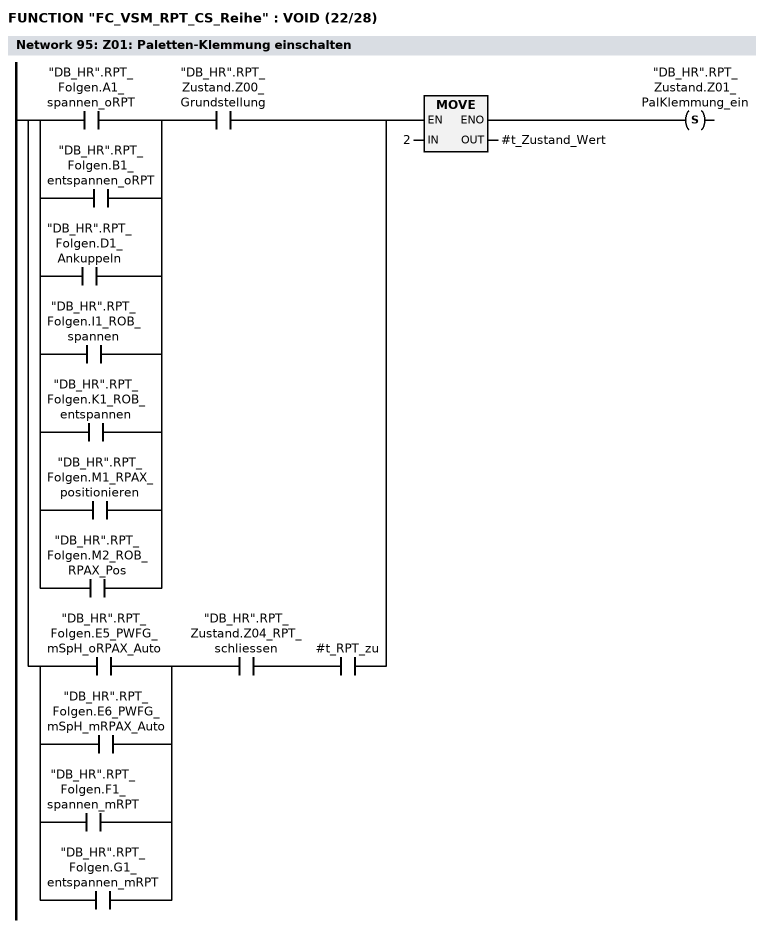

      U(    ;
      U(    ;
      O     "DB_HR".RPT_Folgen.A1_spannen_oRPT;
      O     "DB_HR".RPT_Folgen.B1_entspannen_oRPT;
      O     "DB_HR".RPT_Folgen.D1_Ankuppeln;
      O     "DB_HR".RPT_Folgen.I1_ROB_spannen;
      O     "DB_HR".RPT_Folgen.K1_ROB_entspannen;
      O     "DB_HR".RPT_Folgen.M1_RPAX_positionieren;
//      O     "DB_HR".RPT_Folgen.L2_ROB_PWFG_mRPAX
      O     "DB_HR".RPT_Folgen.M2_ROB_RPAX_Pos;
      )     ;
      U     "DB_HR".RPT_Zustand.Z00_Grundstellung;
      O     ;
      U(    ;
      O     "DB_HR".RPT_Folgen.E5_PWFG_mSpH_oRPAX_Auto;
      O     "DB_HR".RPT_Folgen.E6_PWFG_mSpH_mRPAX_Auto;
      O     "DB_HR".RPT_Folgen.F1_spannen_mRPT;
      O     "DB_HR".RPT_Folgen.G1_entspannen_mRPT;
      )     ;
      U     "DB_HR".RPT_Zustand.Z04_RPT_schliessen;
      U     #t_RPT_zu;
      )     ;
      SPBNB _01d;
      L     2;
      T     #t_Zustand_Wert;
      SET   ;
      SAVE  ;
      CLR   ;
_01d: U     BIE;
      S     "DB_HR".RPT_Zustand.Z01_PalKlemmung_ein;
NETWORK
TITLE =Z02: Ankuppeln
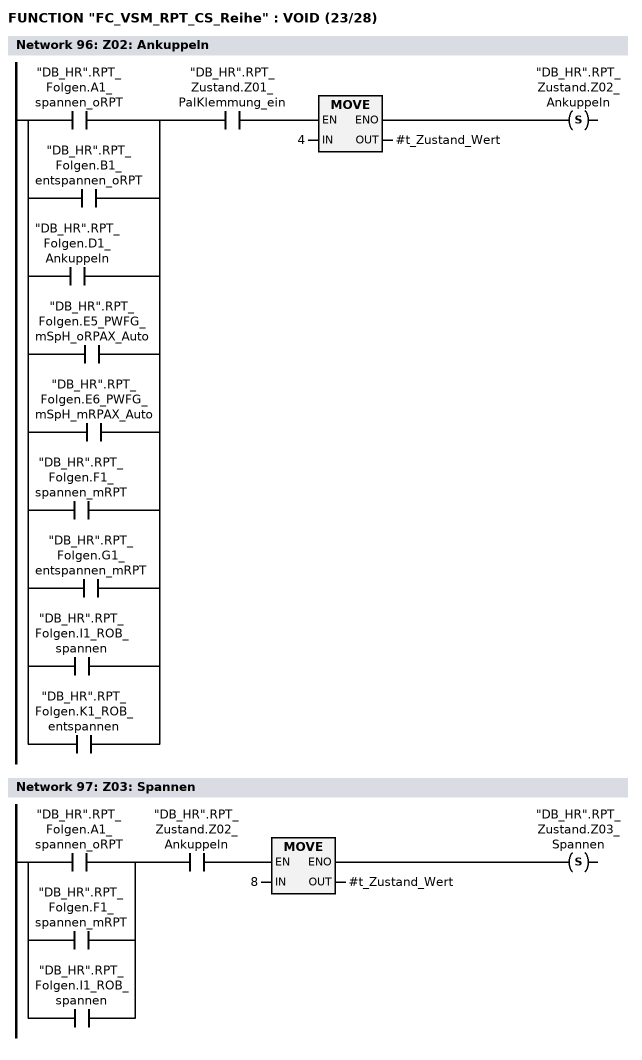

      U(    ;
      O     "DB_HR".RPT_Folgen.A1_spannen_oRPT;
      O     "DB_HR".RPT_Folgen.B1_entspannen_oRPT;
      O     "DB_HR".RPT_Folgen.D1_Ankuppeln;
      O     "DB_HR".RPT_Folgen.E5_PWFG_mSpH_oRPAX_Auto;
      O     "DB_HR".RPT_Folgen.E6_PWFG_mSpH_mRPAX_Auto;
      O     "DB_HR".RPT_Folgen.F1_spannen_mRPT;
      O     "DB_HR".RPT_Folgen.G1_entspannen_mRPT;
      O     "DB_HR".RPT_Folgen.I1_ROB_spannen;
      O     "DB_HR".RPT_Folgen.K1_ROB_entspannen;
      )     ;
      U     "DB_HR".RPT_Zustand.Z01_PalKlemmung_ein;
      SPBNB _01e;
      L     4;
      T     #t_Zustand_Wert;
      SET   ;
      SAVE  ;
      CLR   ;
_01e: U     BIE;
      S     "DB_HR".RPT_Zustand.Z02_Ankuppeln;
NETWORK
TITLE =Z03: Spannen

      U(    ;
      O     "DB_HR".RPT_Folgen.A1_spannen_oRPT;
      O     "DB_HR".RPT_Folgen.F1_spannen_mRPT;
      O     "DB_HR".RPT_Folgen.I1_ROB_spannen;
      )     ;
      U     "DB_HR".RPT_Zustand.Z02_Ankuppeln;
      SPBNB _01f;
      L     8;
      T     #t_Zustand_Wert;
      SET   ;
      SAVE  ;
      CLR   ;
_01f: U     BIE;
      S     "DB_HR".RPT_Zustand.Z03_Spannen;
NETWORK
TITLE =Z04: RPT schließen
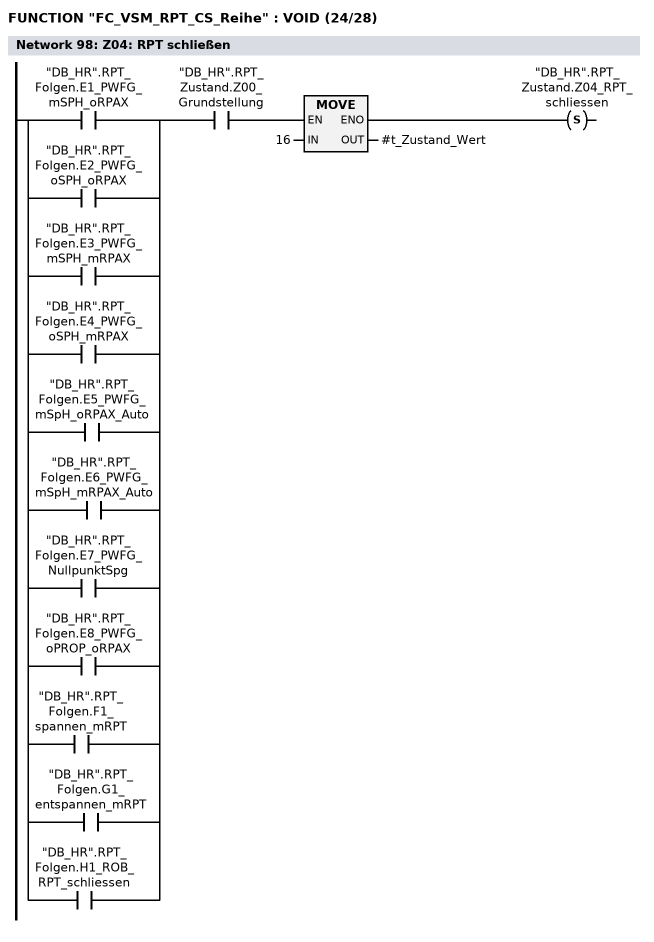

      U(    ;
      O     "DB_HR".RPT_Folgen.E1_PWFG_mSPH_oRPAX;
      O     "DB_HR".RPT_Folgen.E2_PWFG_oSPH_oRPAX;
      O     "DB_HR".RPT_Folgen.E3_PWFG_mSPH_mRPAX;
      O     "DB_HR".RPT_Folgen.E4_PWFG_oSPH_mRPAX;
      O     "DB_HR".RPT_Folgen.E5_PWFG_mSpH_oRPAX_Auto;
      O     "DB_HR".RPT_Folgen.E6_PWFG_mSpH_mRPAX_Auto;
      O     "DB_HR".RPT_Folgen.E7_PWFG_NullpunktSpg;
      O     "DB_HR".RPT_Folgen.E8_PWFG_oPROP_oRPAX;
      O     "DB_HR".RPT_Folgen.F1_spannen_mRPT;
      O     "DB_HR".RPT_Folgen.G1_entspannen_mRPT;
      O     "DB_HR".RPT_Folgen.H1_ROB_RPT_schliessen;
      )     ;
      U     "DB_HR".RPT_Zustand.Z00_Grundstellung;
      SPBNB _020;
      L     16;
      T     #t_Zustand_Wert;
      SET   ;
      SAVE  ;
      CLR   ;
_020: U     BIE;
      S     "DB_HR".RPT_Zustand.Z04_RPT_schliessen;
NETWORK
TITLE =Z05: Abkuppeln
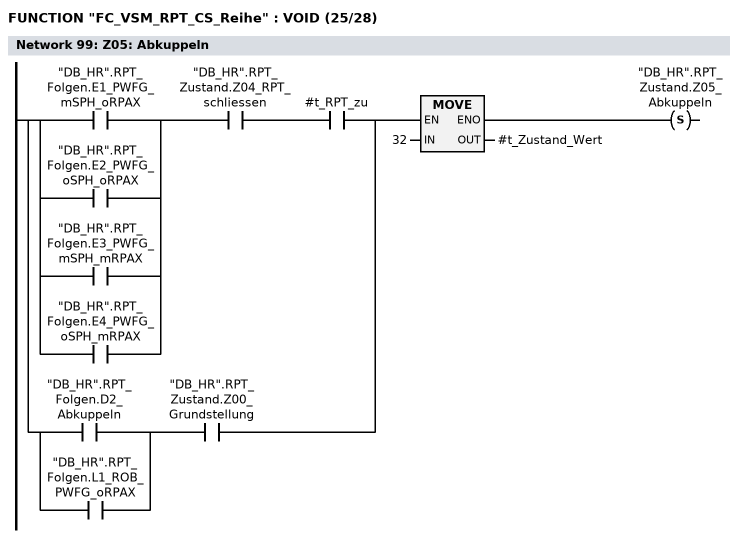

      U(    ;
      U(    ;
      O     "DB_HR".RPT_Folgen.E1_PWFG_mSPH_oRPAX;
      O     "DB_HR".RPT_Folgen.E2_PWFG_oSPH_oRPAX;
      O     "DB_HR".RPT_Folgen.E3_PWFG_mSPH_mRPAX;
      O     "DB_HR".RPT_Folgen.E4_PWFG_oSPH_mRPAX;
      )     ;
      U     "DB_HR".RPT_Zustand.Z04_RPT_schliessen;
      U     #t_RPT_zu;
      O     ;
      U(    ;
      O     "DB_HR".RPT_Folgen.D2_Abkuppeln;
      O     "DB_HR".RPT_Folgen.L1_ROB_PWFG_oRPAX;
      )     ;
      U     "DB_HR".RPT_Zustand.Z00_Grundstellung;
      )     ;
      SPBNB _021;
      L     32;
      T     #t_Zustand_Wert;
      SET   ;
      SAVE  ;
      CLR   ;
_021: U     BIE;
      S     "DB_HR".RPT_Zustand.Z05_Abkuppeln;
NETWORK
TITLE =Z07: PW-Freigabe aktivieren
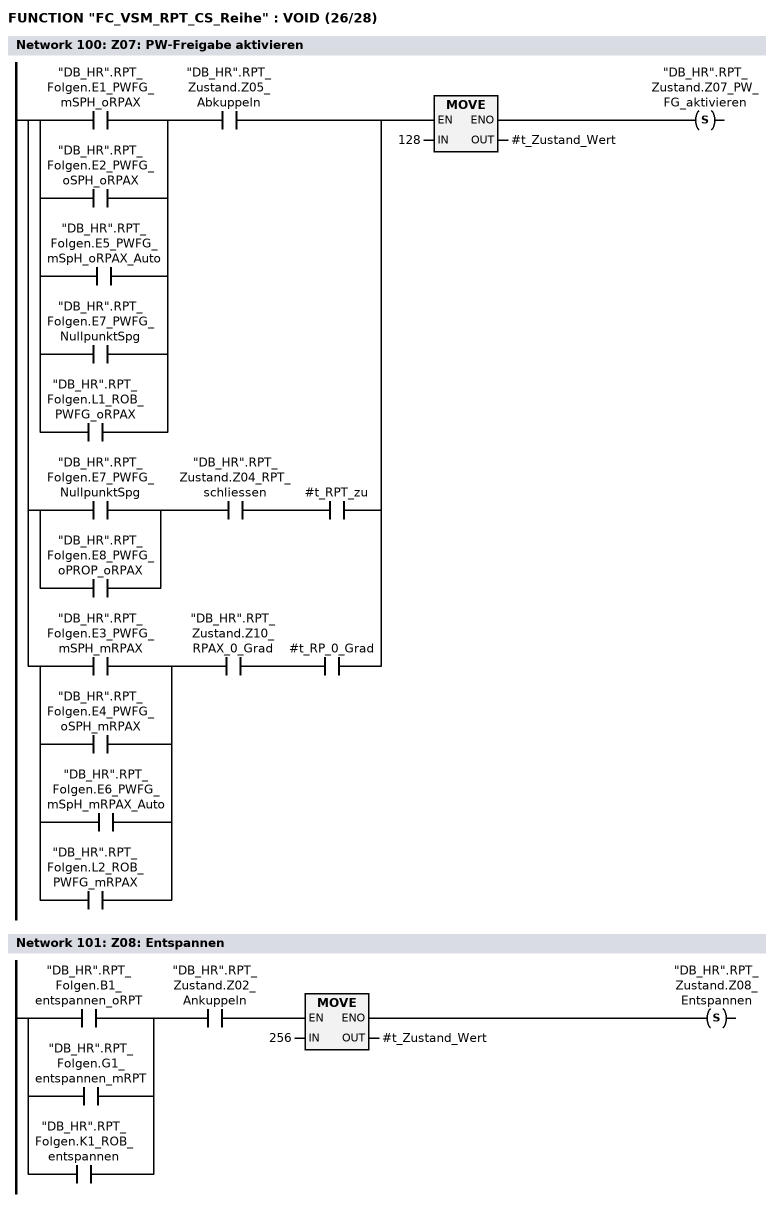

      U(    ;
      U(    ;
      O     "DB_HR".RPT_Folgen.E1_PWFG_mSPH_oRPAX;
      O     "DB_HR".RPT_Folgen.E2_PWFG_oSPH_oRPAX;
      O     "DB_HR".RPT_Folgen.E5_PWFG_mSpH_oRPAX_Auto;
      O     "DB_HR".RPT_Folgen.E7_PWFG_NullpunktSpg;
      O     "DB_HR".RPT_Folgen.L1_ROB_PWFG_oRPAX;
      )     ;
      U     "DB_HR".RPT_Zustand.Z05_Abkuppeln;
      O     ;
      U(    ;
      O     "DB_HR".RPT_Folgen.E7_PWFG_NullpunktSpg;
      O     "DB_HR".RPT_Folgen.E8_PWFG_oPROP_oRPAX;
      )     ;
      U     "DB_HR".RPT_Zustand.Z04_RPT_schliessen;
      U     #t_RPT_zu;
      O     ;
      U(    ;
      O     "DB_HR".RPT_Folgen.E3_PWFG_mSPH_mRPAX;
      O     "DB_HR".RPT_Folgen.E4_PWFG_oSPH_mRPAX;
      O     "DB_HR".RPT_Folgen.E6_PWFG_mSpH_mRPAX_Auto;
      O     "DB_HR".RPT_Folgen.L2_ROB_PWFG_mRPAX;
      )     ;
      U     "DB_HR".RPT_Zustand.Z10_RPAX_0_Grad;
      U     #t_RP_0_Grad;
      )     ;
      SPBNB _022;
      L     128;
      T     #t_Zustand_Wert;
      SET   ;
      SAVE  ;
      CLR   ;
_022: U     BIE;
      S     "DB_HR".RPT_Zustand.Z07_PW_FG_aktivieren;
NETWORK
TITLE =Z08: Entspannen

      U(    ;
      O     "DB_HR".RPT_Folgen.B1_entspannen_oRPT;
      O     "DB_HR".RPT_Folgen.G1_entspannen_mRPT;
      O     "DB_HR".RPT_Folgen.K1_ROB_entspannen;
      )     ;
      U     "DB_HR".RPT_Zustand.Z02_Ankuppeln;
      SPBNB _023;
      L     256;
      T     #t_Zustand_Wert;
      SET   ;
      SAVE  ;
      CLR   ;
_023: U     BIE;
      S     "DB_HR".RPT_Zustand.Z08_Entspannen;
NETWORK
TITLE =Z09: RPT öffnen
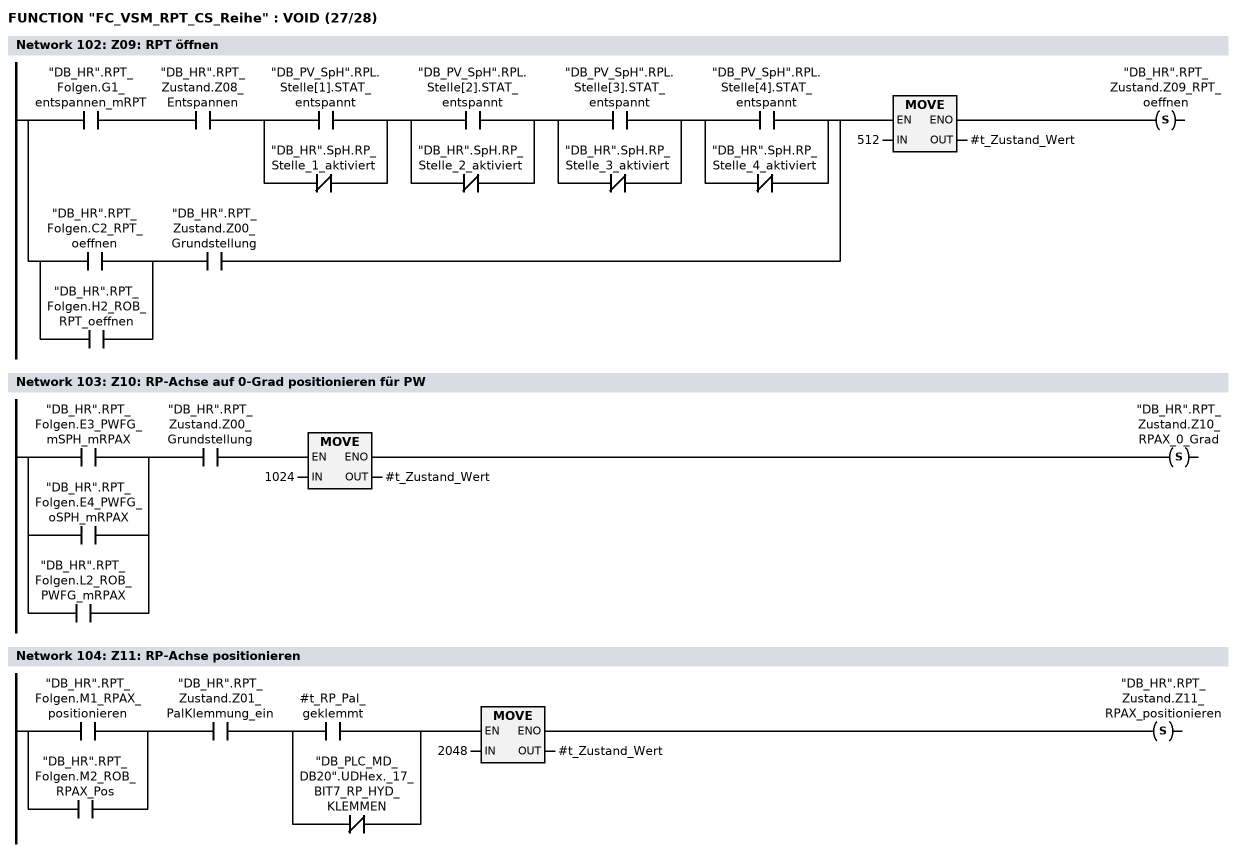

      U(    ;
      U     "DB_HR".RPT_Folgen.G1_entspannen_mRPT;
      U     "DB_HR".RPT_Zustand.Z08_Entspannen;
      U(    ;
      O     "DB_PV_SpH".RPL.Stelle[1].STAT_entspannt;
      ON    "DB_HR".SpH.RP_Stelle_1_aktiviert;
      )     ;
      U(    ;
      O     "DB_PV_SpH".RPL.Stelle[2].STAT_entspannt;
      ON    "DB_HR".SpH.RP_Stelle_2_aktiviert;
      )     ;
      U(    ;
      O     "DB_PV_SpH".RPL.Stelle[3].STAT_entspannt;
      ON    "DB_HR".SpH.RP_Stelle_3_aktiviert;
      )     ;
      U(    ;
      O     "DB_PV_SpH".RPL.Stelle[4].STAT_entspannt;
      ON    "DB_HR".SpH.RP_Stelle_4_aktiviert;
      )     ;
      O     ;
      U(    ;
      O     "DB_HR".RPT_Folgen.C2_RPT_oeffnen;
      O     "DB_HR".RPT_Folgen.H2_ROB_RPT_oeffnen;
      )     ;
      U     "DB_HR".RPT_Zustand.Z00_Grundstellung;
      )     ;
      SPBNB _024;
      L     512;
      T     #t_Zustand_Wert;
      SET   ;
      SAVE  ;
      CLR   ;
_024: U     BIE;
      S     "DB_HR".RPT_Zustand.Z09_RPT_oeffnen;
NETWORK
TITLE =Z10: RP-Achse auf 0-Grad positionieren für PW

      U(    ;
      O     "DB_HR".RPT_Folgen.E3_PWFG_mSPH_mRPAX;
      O     "DB_HR".RPT_Folgen.E4_PWFG_oSPH_mRPAX;
      O     "DB_HR".RPT_Folgen.L2_ROB_PWFG_mRPAX;
      )     ;
//      U     "DB_HR".RPT_Zustand.Z05_Abkuppeln
      U     "DB_HR".RPT_Zustand.Z00_Grundstellung;
      SPBNB _025;
      L     1024;
      T     #t_Zustand_Wert;
      SET   ;
      SAVE  ;
      CLR   ;
_025: U     BIE;
      S     "DB_HR".RPT_Zustand.Z10_RPAX_0_Grad;
NETWORK
TITLE =Z11: RP-Achse positionieren

      U(    ;
      O     "DB_HR".RPT_Folgen.M1_RPAX_positionieren;
      O     "DB_HR".RPT_Folgen.M2_ROB_RPAX_Pos;
      )     ;
      U     "DB_HR".RPT_Zustand.Z01_PalKlemmung_ein;
      U(    ;
      O     #t_RP_Pal_geklemmt;
      ON    "DB_PLC_MD_DB20".UDHex._17_BIT7_RP_HYD_KLEMMEN;
      )     ;
      SPBNB _026;
      L     2048;
      T     #t_Zustand_Wert;
      SET   ;
      SAVE  ;
      CLR   ;
_026: U     BIE;
      S     "DB_HR".RPT_Zustand.Z11_RPAX_positionieren;
NETWORK
TITLE =Z15: Abbruch
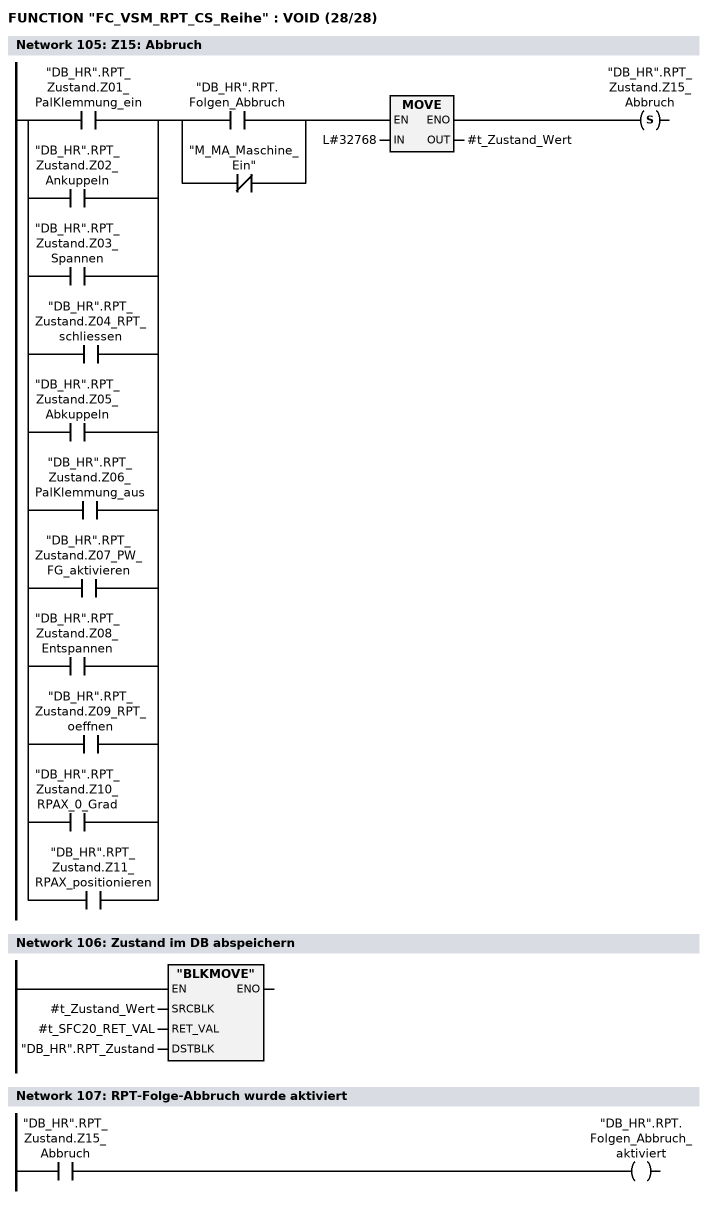

      U(    ;
      O     "DB_HR".RPT_Zustand.Z01_PalKlemmung_ein;
      O     "DB_HR".RPT_Zustand.Z02_Ankuppeln;
      O     "DB_HR".RPT_Zustand.Z03_Spannen;
      O     "DB_HR".RPT_Zustand.Z04_RPT_schliessen;
      O     "DB_HR".RPT_Zustand.Z05_Abkuppeln;
      O     "DB_HR".RPT_Zustand.Z06_PalKlemmung_aus;
      O     "DB_HR".RPT_Zustand.Z07_PW_FG_aktivieren;
      O     "DB_HR".RPT_Zustand.Z08_Entspannen;
      O     "DB_HR".RPT_Zustand.Z09_RPT_oeffnen;
      O     "DB_HR".RPT_Zustand.Z10_RPAX_0_Grad;
      O     "DB_HR".RPT_Zustand.Z11_RPAX_positionieren;
      )     ;
      U(    ;
      O     "DB_HR".RPT.Folgen_Abbruch;
      ON    "M_MA_Maschine_Ein";
      )     ;
      SPBNB _027;
      L     L#32768;
      T     #t_Zustand_Wert;
      SET   ;
      SAVE  ;
      CLR   ;
_027: U     BIE;
      S     "DB_HR".RPT_Zustand.Z15_Abbruch;
NETWORK
TITLE =Zustand im DB abspeichern

      CALL "BLKMOVE" (
           SRCBLK                   := #t_Zustand_Wert,
           RET_VAL                  := #t_SFC20_RET_VAL,
           DSTBLK                   := "DB_HR".RPT_Zustand);
      NOP   0;
NETWORK
TITLE =RPT-Folge-Abbruch wurde aktiviert

      U     "DB_HR".RPT_Zustand.Z15_Abbruch;
      =     "DB_HR".RPT.Folgen_Abbruch_aktiviert;
NETWORK
TITLE =Freigabe RPT-Tür-Zylinder öffnen

      U(    ;
      U(    ;
      U(    ;
      O     "DB_HR".RPT_Zustand.Z09_RPT_oeffnen;
      O     "DB_EINRICHTFUNKTION".Bewegung_38_Minus;
      )     ;
      U(    ;
      O     #t_RPT_zu;
      ON    #t_RPT_zu;
      )     ;
      O     ;
      U     "DB_HR".ROB_Interface.PI_SS_Roboter;
      U     "DB_OUT".AmxSusDoorOpen;
      )     ;
      S     "DB_HR".RPT.FG_TuerZyl_oeffnen;
      U(    ;
      O     "DB_HR".RPT_Zustand.Z04_RPT_schliessen;
      O     "DB_EINRICHTFUNKTION".Bewegung_38_Plus;
      O     ;
      U     "DB_HR".ROB_Interface.PI_SS_Roboter;
      U     #t_RPT_zu;
      )     ;
      R     "DB_HR".RPT.FG_TuerZyl_oeffnen;
      U     "DB_HR".RPT.FG_TuerZyl_oeffnen;
      )     ;
      U     "DB_HR".ABST.Automatische_RPT;
      =     "DB_IN".ImxOpenSusDoor;
NETWORK
TITLE =Freigabe RPT-Tür-Zylinder schließen

      U(    ;
      U(    ;
      O     "DB_HR".RPT_Zustand.Z04_RPT_schliessen;
      O     "DB_EINRICHTFUNKTION".Bewegung_38_Plus;
      O     ;
      U     "DB_HR".ROB_Interface.PI_SS_Roboter;
      U     #t_RPT_zu;
      )     ;
      S     "DB_HR".RPT.FG_TuerZyl_schliessen;
      U(    ;
      O     "DB_HR".RPT_Zustand.Z09_RPT_oeffnen;
      O     "DB_EINRICHTFUNKTION".Bewegung_38_Minus;
      O     ;
      U     "DB_HR".ROB_Interface.PI_SS_Roboter;
      U     "DB_OUT".AmxSusDoorOpen;
      )     ;
      R     "DB_HR".RPT.FG_TuerZyl_schliessen;
      U     "DB_HR".RPT.FG_TuerZyl_schliessen;
      )     ;
      U     "DB_HR".ABST.Automatische_RPT;
      =     "DB_IN".ImxCloseSusDoor;
NETWORK
TITLE =Merker eine SpannHydraulik-Spann-Folge ist aktiv
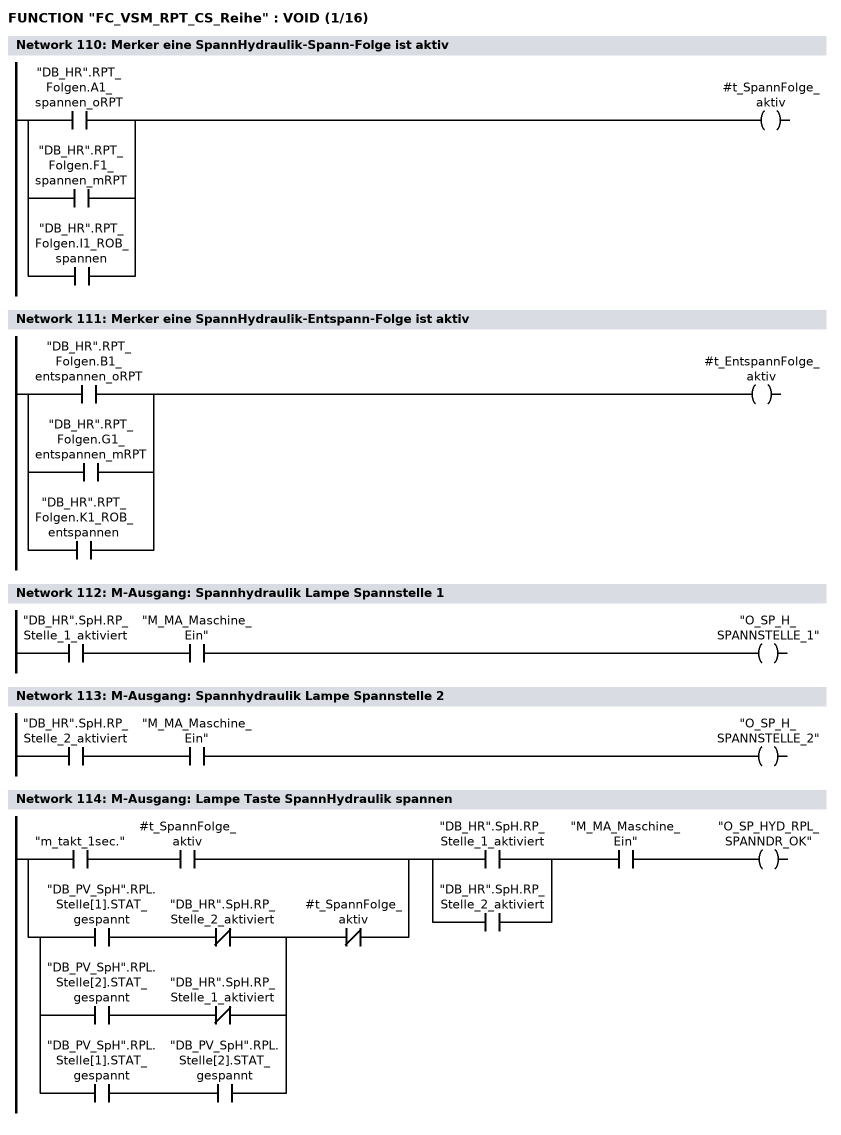

      O     "DB_HR".RPT_Folgen.A1_spannen_oRPT;
      O     "DB_HR".RPT_Folgen.F1_spannen_mRPT;
      O     "DB_HR".RPT_Folgen.I1_ROB_spannen;
      =     #t_SpannFolge_aktiv;
NETWORK
TITLE =Merker eine SpannHydraulik-Entspann-Folge ist aktiv

      O     "DB_HR".RPT_Folgen.B1_entspannen_oRPT;
      O     "DB_HR".RPT_Folgen.G1_entspannen_mRPT;
      O     "DB_HR".RPT_Folgen.K1_ROB_entspannen;
      =     #t_EntspannFolge_aktiv;
NETWORK
TITLE =M-Ausgang: Spannhydraulik Lampe Spannstelle 1

      U     "DB_HR".SpH.RP_Stelle_1_aktiviert;
      U     "M_MA_Maschine_Ein";
      =     "O_SP_H_SPANNSTELLE_1";
NETWORK
TITLE =M-Ausgang: Spannhydraulik Lampe Spannstelle 2

      U     "DB_HR".SpH.RP_Stelle_2_aktiviert;
      U     "M_MA_Maschine_Ein";
      =     "O_SP_H_SPANNSTELLE_2";
NETWORK
TITLE =M-Ausgang: Lampe Taste SpannHydraulik spannen

      U(    ;
      U     "m_takt_1sec.";
      U     #t_SpannFolge_aktiv;
      O     ;
      U(    ;
      U     "DB_PV_SpH".RPL.Stelle[1].STAT_gespannt;
      UN    "DB_HR".SpH.RP_Stelle_2_aktiviert;
      O     ;
      U     "DB_PV_SpH".RPL.Stelle[2].STAT_gespannt;
      UN    "DB_HR".SpH.RP_Stelle_1_aktiviert;
      O     ;
      U     "DB_PV_SpH".RPL.Stelle[1].STAT_gespannt;
      U     "DB_PV_SpH".RPL.Stelle[2].STAT_gespannt;
      )     ;
      UN    #t_SpannFolge_aktiv;
      )     ;
      U(    ;
      O     "DB_HR".SpH.RP_Stelle_1_aktiviert;
      O     "DB_HR".SpH.RP_Stelle_2_aktiviert;
      )     ;
      U     "M_MA_Maschine_Ein";
      =     "O_SP_HYD_RPL_SPANNDR_OK";
NETWORK
TITLE =M-Ausgang: Lampe Taste SpannHydraulik entspannen
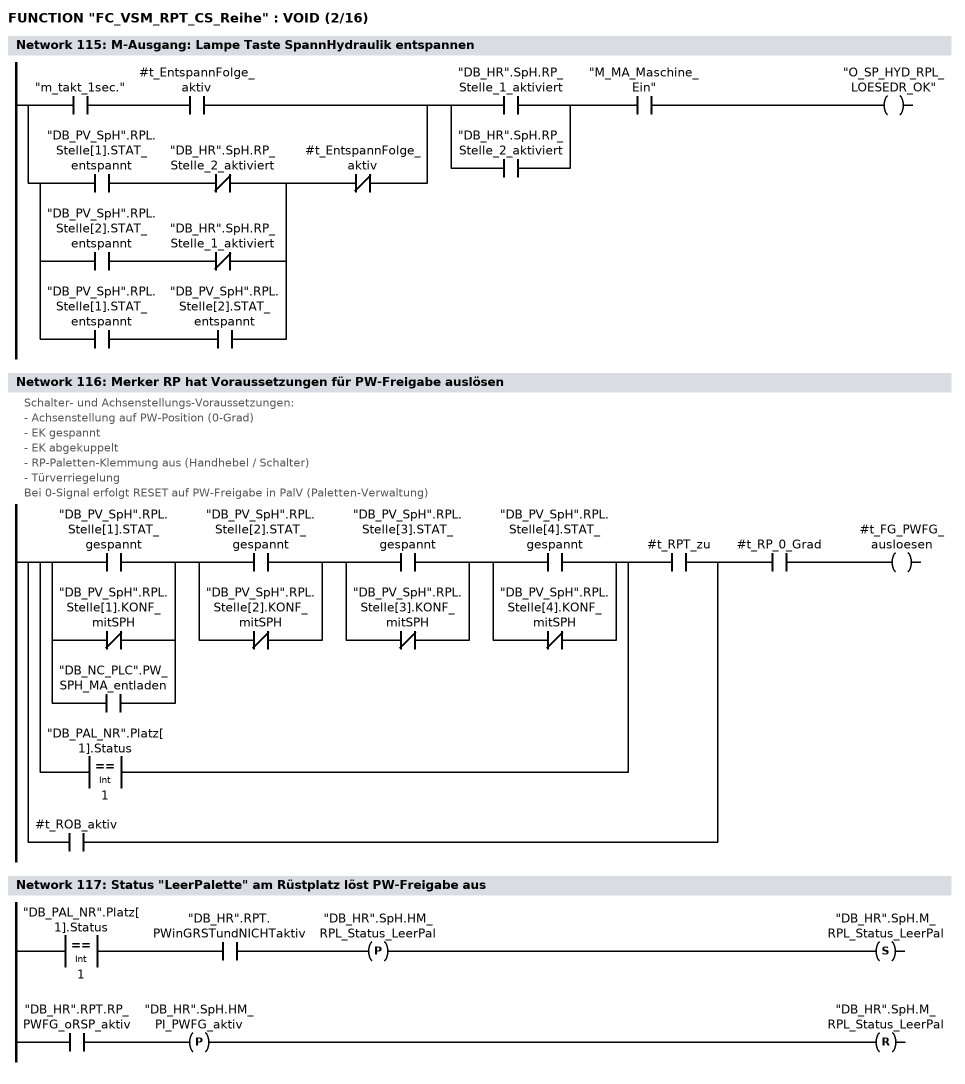

      U(    ;
      U     "m_takt_1sec.";
      U     #t_EntspannFolge_aktiv;
      O     ;
      U(    ;
      U     "DB_PV_SpH".RPL.Stelle[1].STAT_entspannt;
      UN    "DB_HR".SpH.RP_Stelle_2_aktiviert;
      O     ;
      U     "DB_PV_SpH".RPL.Stelle[2].STAT_entspannt;
      UN    "DB_HR".SpH.RP_Stelle_1_aktiviert;
      O     ;
      U     "DB_PV_SpH".RPL.Stelle[1].STAT_entspannt;
      U     "DB_PV_SpH".RPL.Stelle[2].STAT_entspannt;
      )     ;
      UN    #t_EntspannFolge_aktiv;
      )     ;
      U(    ;
      O     "DB_HR".SpH.RP_Stelle_1_aktiviert;
      O     "DB_HR".SpH.RP_Stelle_2_aktiviert;
      )     ;
      U     "M_MA_Maschine_Ein";
      =     "O_SP_HYD_RPL_LOESEDR_OK";
NETWORK
TITLE =Merker RP hat Voraussetzungen für PW-Freigabe auslösen
//Schalter- und Achsenstellungs-Voraussetzungen:
//- Achsenstellung auf PW-Position (0-Grad)
//- EK gespannt
//- EK abgekuppelt
//- RP-Paletten-Klemmung aus (Handhebel / Schalter)
//- Türverriegelung
//
//Bei 0-Signal erfolgt RESET auf PW-Freigabe in PalV (Paletten-Verwaltung)
      U(    ;
      U(    ;
      U(    ;
      O     "DB_PV_SpH".RPL.Stelle[1].STAT_gespannt;
      ON    "DB_PV_SpH".RPL.Stelle[1].KONF_mitSPH;
      O     "DB_NC_PLC".PW_SPH_MA_entladen;
      )     ;
      U(    ;
      O     "DB_PV_SpH".RPL.Stelle[2].STAT_gespannt;
      ON    "DB_PV_SpH".RPL.Stelle[2].KONF_mitSPH;
      )     ;
      U(    ;
      O     "DB_PV_SpH".RPL.Stelle[3].STAT_gespannt;
      ON    "DB_PV_SpH".RPL.Stelle[3].KONF_mitSPH;
      )     ;
      U(    ;
      O     "DB_PV_SpH".RPL.Stelle[4].STAT_gespannt;
      ON    "DB_PV_SpH".RPL.Stelle[4].KONF_mitSPH;
      )     ;
      O(    ;
      L     "DB_PAL_NR".Platz[1].Status;
      L     1;
      ==I   ;
      )     ;
      )     ;
      U     #t_RPT_zu;
      O     #t_ROB_aktiv;
      )     ;
      U     #t_RP_0_Grad;
      =     #t_FG_PWFG_ausloesen;
NETWORK
TITLE =Status "LeerPalette" am Rüstplatz löst PW-Freigabe aus

      U(    ;
      L     "DB_PAL_NR".Platz[1].Status;
      L     1;
      ==I   ;
      )     ;
      U     "DB_HR".RPT.PWinGRSTundNICHTaktiv;
      FP    "DB_HR".SpH.HM_RPL_Status_LeerPal;
      S     "DB_HR".SpH.M_RPL_Status_LeerPal;
      U     "DB_HR".RPT.RP_PWFG_oRSP_aktiv;
      FP    "DB_HR".SpH.HM_PI_PWFG_aktiv;
      R     "DB_HR".SpH.M_RPL_Status_LeerPal;
      NOP   0;
NETWORK
TITLE =PW-Freigabe OHNE Rundspeicher ist aktiv
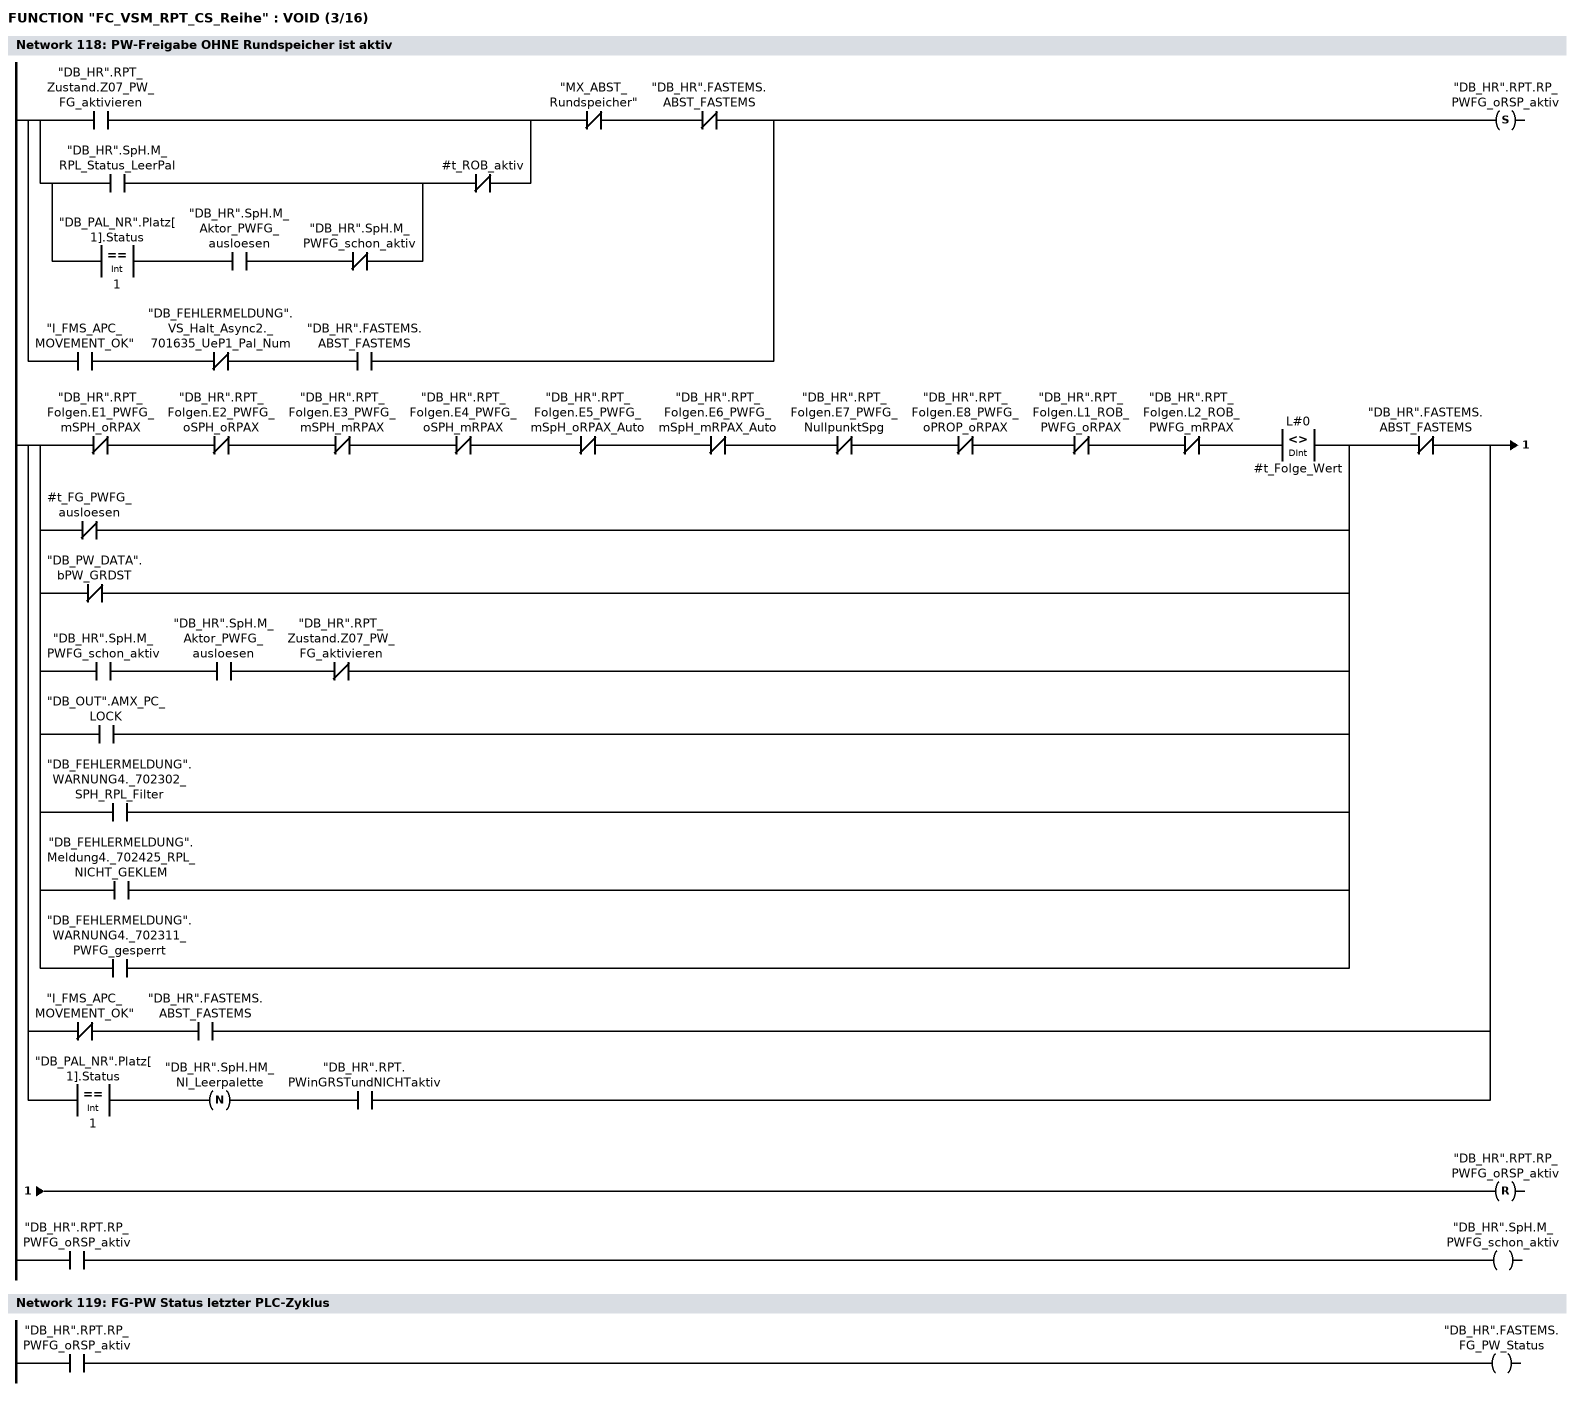

      U(    ;
      U(    ;
      O     "DB_HR".RPT_Zustand.Z07_PW_FG_aktivieren;
      O     ;
      U(    ;
      O     "DB_HR".SpH.M_RPL_Status_LeerPal;
      O     ;
      U(    ;
      L     "DB_PAL_NR".Platz[1].Status;
      L     1;
      ==I   ;
      )     ;
      U     "DB_HR".SpH.M_Aktor_PWFG_ausloesen;
      UN    "DB_HR".SpH.M_PWFG_schon_aktiv;
      )     ;
      UN    #t_ROB_aktiv;
      )     ;
      UN    "MX_ABST_Rundspeicher";
      UN    "DB_HR".FASTEMS.ABST_FASTEMS;
      O     ;
      U     "I_FMS_APC_MOVEMENT_OK";
      UN    "DB_FEHLERMELDUNG".VS_Halt_Async2._701635_UeP1_Pal_Num;
      U     "DB_HR".FASTEMS.ABST_FASTEMS;
      )     ;
      S     "DB_HR".RPT.RP_PWFG_oRSP_aktiv;
      U(    ;
      U(    ;
      UN    "DB_HR".RPT_Folgen.E1_PWFG_mSPH_oRPAX;
      UN    "DB_HR".RPT_Folgen.E2_PWFG_oSPH_oRPAX;
      UN    "DB_HR".RPT_Folgen.E3_PWFG_mSPH_mRPAX;
      UN    "DB_HR".RPT_Folgen.E4_PWFG_oSPH_mRPAX;
      UN    "DB_HR".RPT_Folgen.E5_PWFG_mSpH_oRPAX_Auto;
      UN    "DB_HR".RPT_Folgen.E6_PWFG_mSpH_mRPAX_Auto;
      UN    "DB_HR".RPT_Folgen.E7_PWFG_NullpunktSpg;
      UN    "DB_HR".RPT_Folgen.E8_PWFG_oPROP_oRPAX;
      UN    "DB_HR".RPT_Folgen.L1_ROB_PWFG_oRPAX;
      UN    "DB_HR".RPT_Folgen.L2_ROB_PWFG_mRPAX;
      U(    ;
      L     L#0;
      L     #t_Folge_Wert;
      <>D   ;
      )     ;
      ON    #t_FG_PWFG_ausloesen;
      ON    "DB_PW_DATA".bPW_GRDST;
      O     ;
      U     "DB_HR".SpH.M_PWFG_schon_aktiv;
      U     "DB_HR".SpH.M_Aktor_PWFG_ausloesen;
      UN    "DB_HR".RPT_Zustand.Z07_PW_FG_aktivieren;
      O     "DB_OUT".AMX_PC_LOCK;
      O     "DB_FEHLERMELDUNG".WARNUNG4._702302_SPH_RPL_Filter;
      O     "DB_FEHLERMELDUNG".Meldung4._702425_RPL_NICHT_GEKLEM;
      O     "DB_FEHLERMELDUNG".WARNUNG4._702311_PWFG_gesperrt;
      )     ;
      UN    "DB_HR".FASTEMS.ABST_FASTEMS;
      O(    ;
      UN    "I_FMS_APC_MOVEMENT_OK";
      U     "DB_HR".FASTEMS.ABST_FASTEMS;
      )     ;
      O(    ;
      U(    ;
      L     "DB_PAL_NR".Platz[1].Status;
      L     1;
      ==I   ;
      )     ;
      FN    "DB_HR".SpH.HM_NI_Leerpalette;
      U     "DB_HR".RPT.PWinGRSTundNICHTaktiv;
      )     ;
      )     ;
      R     "DB_HR".RPT.RP_PWFG_oRSP_aktiv;
      U     "DB_HR".RPT.RP_PWFG_oRSP_aktiv;
      =     "DB_HR".SpH.M_PWFG_schon_aktiv;
NETWORK
TITLE =FG-PW Status letzter PLC-Zyklus

      U     "DB_HR".RPT.RP_PWFG_oRSP_aktiv;
      =     "DB_HR".FASTEMS.FG_PW_Status;
NETWORK
TITLE =VSM-intern Freigabe Palette am RPL-Rundspeicher
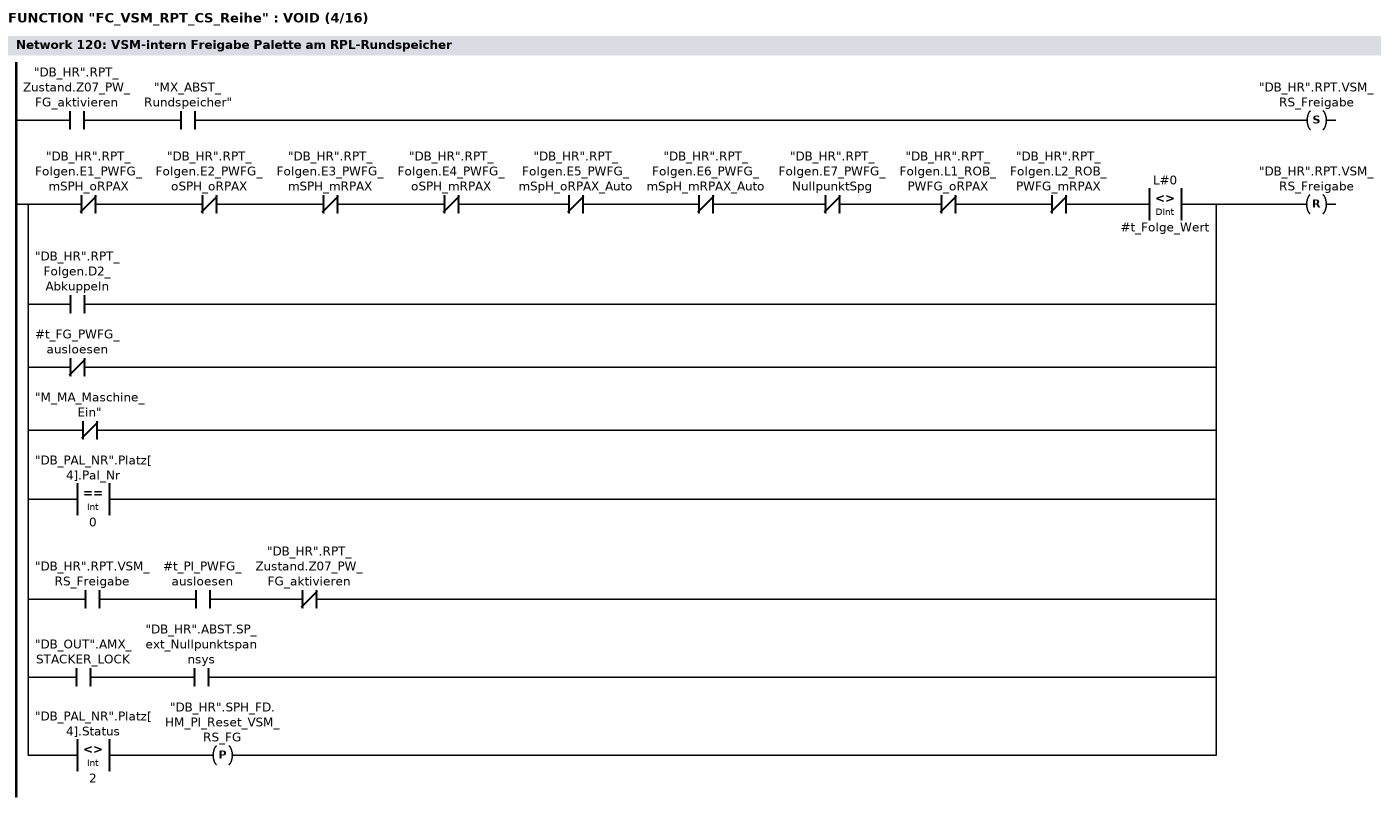

      U     "DB_HR".RPT_Zustand.Z07_PW_FG_aktivieren;
      U     "MX_ABST_Rundspeicher";
      S     "DB_HR".RPT.VSM_RS_Freigabe;
      U(    ;
      UN    "DB_HR".RPT_Folgen.E1_PWFG_mSPH_oRPAX;
      UN    "DB_HR".RPT_Folgen.E2_PWFG_oSPH_oRPAX;
      UN    "DB_HR".RPT_Folgen.E3_PWFG_mSPH_mRPAX;
      UN    "DB_HR".RPT_Folgen.E4_PWFG_oSPH_mRPAX;
      UN    "DB_HR".RPT_Folgen.E5_PWFG_mSpH_oRPAX_Auto;
      UN    "DB_HR".RPT_Folgen.E6_PWFG_mSpH_mRPAX_Auto;
      UN    "DB_HR".RPT_Folgen.E7_PWFG_NullpunktSpg;
      UN    "DB_HR".RPT_Folgen.L1_ROB_PWFG_oRPAX;
      UN    "DB_HR".RPT_Folgen.L2_ROB_PWFG_mRPAX;
      U(    ;
      L     L#0;
      L     #t_Folge_Wert;
      <>D   ;
      )     ;
      O     "DB_HR".RPT_Folgen.D2_Abkuppeln;
      ON    #t_FG_PWFG_ausloesen;
      ON    "M_MA_Maschine_Ein";
      O(    ;
      L     "DB_PAL_NR".Platz[4].Pal_Nr;
      L     0;
      ==I   ;
      )     ;
      O(    ;
      U     "DB_HR".RPT.VSM_RS_Freigabe;
      U     #t_PI_PWFG_ausloesen;
      UN    "DB_HR".RPT_Zustand.Z07_PW_FG_aktivieren;
      )     ;
      O(    ;
      U     "DB_OUT".AMX_STACKER_LOCK;
      U     "DB_HR".ABST.SP_ext_Nullpunktspannsys;
      )     ;
      O(    ;
      U(    ;
      L     "DB_PAL_NR".Platz[4].Status;
      L     2;
      <>I   ;
      )     ;
      FP    "DB_HR".SPH_FD.HM_PI_Reset_VSM_RS_FG;
      )     ;
      )     ;
      R     "DB_HR".RPT.VSM_RS_Freigabe;
      NOP   0;
NETWORK
TITLE =M-Ausgang: Lampe Taste PW Freigabe
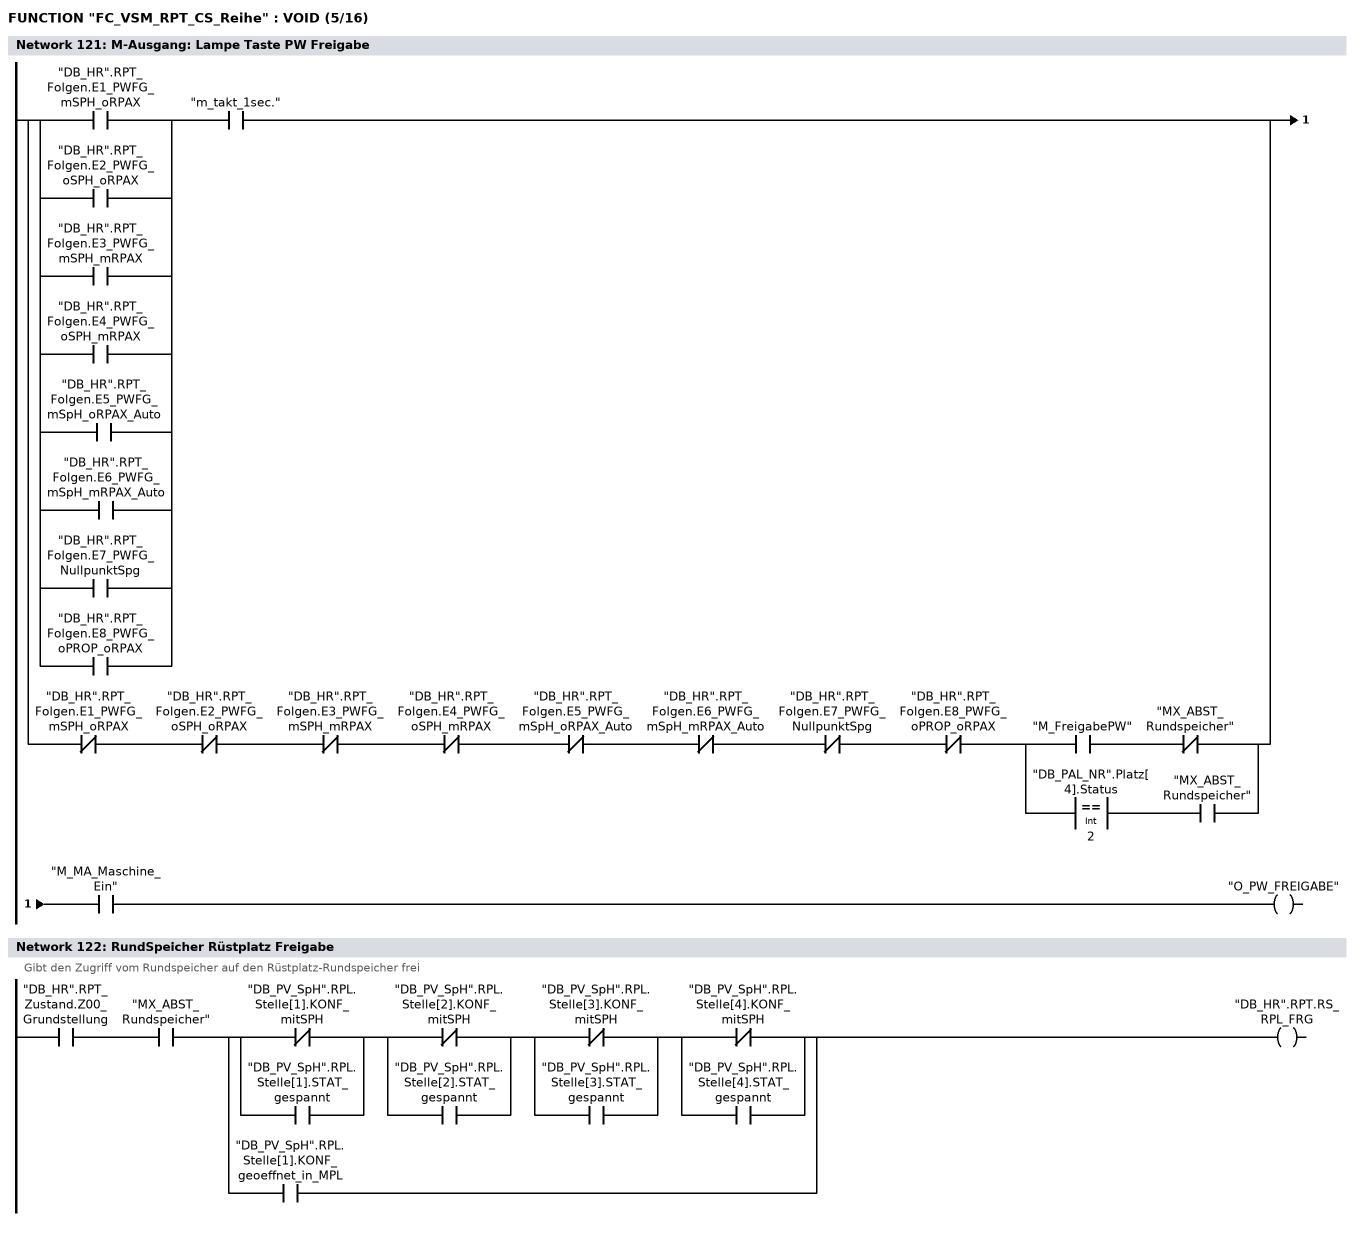

      U(    ;
      U(    ;
      O     "DB_HR".RPT_Folgen.E1_PWFG_mSPH_oRPAX;
      O     "DB_HR".RPT_Folgen.E2_PWFG_oSPH_oRPAX;
      O     "DB_HR".RPT_Folgen.E3_PWFG_mSPH_mRPAX;
      O     "DB_HR".RPT_Folgen.E4_PWFG_oSPH_mRPAX;
      O     "DB_HR".RPT_Folgen.E5_PWFG_mSpH_oRPAX_Auto;
      O     "DB_HR".RPT_Folgen.E6_PWFG_mSpH_mRPAX_Auto;
      O     "DB_HR".RPT_Folgen.E7_PWFG_NullpunktSpg;
      O     "DB_HR".RPT_Folgen.E8_PWFG_oPROP_oRPAX;
      )     ;
      U     "m_takt_1sec.";
      O     ;
      UN    "DB_HR".RPT_Folgen.E1_PWFG_mSPH_oRPAX;
      UN    "DB_HR".RPT_Folgen.E2_PWFG_oSPH_oRPAX;
      UN    "DB_HR".RPT_Folgen.E3_PWFG_mSPH_mRPAX;
      UN    "DB_HR".RPT_Folgen.E4_PWFG_oSPH_mRPAX;
      UN    "DB_HR".RPT_Folgen.E5_PWFG_mSpH_oRPAX_Auto;
      UN    "DB_HR".RPT_Folgen.E6_PWFG_mSpH_mRPAX_Auto;
      UN    "DB_HR".RPT_Folgen.E7_PWFG_NullpunktSpg;
      UN    "DB_HR".RPT_Folgen.E8_PWFG_oPROP_oRPAX;
      U(    ;
      U     "M_FreigabePW";
      UN    "MX_ABST_Rundspeicher";
      O     ;
      U(    ;
      L     "DB_PAL_NR".Platz[4].Status;
      L     2;
      ==I   ;
      )     ;
      U     "MX_ABST_Rundspeicher";
      )     ;
      )     ;
      U     "M_MA_Maschine_Ein";
      =     "O_PW_FREIGABE";

NETWORK
TITLE =RundSpeicher Rüstplatz Freigabe
//Gibt den Zugriff vom Rundspeicher auf den Rüstplatz-Rundspeicher frei
      U     "DB_HR".RPT_Zustand.Z00_Grundstellung;
      U     "MX_ABST_Rundspeicher";
      U(    ;
      U(    ;
      ON    "DB_PV_SpH".RPL.Stelle[1].KONF_mitSPH;
      O     "DB_PV_SpH".RPL.Stelle[1].STAT_gespannt;
      )     ;
      U(    ;
      ON    "DB_PV_SpH".RPL.Stelle[2].KONF_mitSPH;
      O     "DB_PV_SpH".RPL.Stelle[2].STAT_gespannt;
      )     ;
      U(    ;
      ON    "DB_PV_SpH".RPL.Stelle[3].KONF_mitSPH;
      O     "DB_PV_SpH".RPL.Stelle[3].STAT_gespannt;
      )     ;
      U(    ;
      ON    "DB_PV_SpH".RPL.Stelle[4].KONF_mitSPH;
      O     "DB_PV_SpH".RPL.Stelle[4].STAT_gespannt;
      )     ;
      O     "DB_PV_SpH".RPL.Stelle[1].KONF_geoeffnet_in_MPL;
      )     ;
      =     "DB_HR".RPT.RS_RPL_FRG;
NETWORK
TITLE =M-AUSGANG: Rückschlagventil Entspann-Leitung RPL öffnen
//Wenn das Ventil bestromt ist, ist der Entspanndruck eingesperrt.
//Damit sicher gestellt ist, dass beim Umrüsten einer Palette am Rüstplatz, der
//eingesperrte Druck auf der Entspannseite entweichen kann,
//erfolgt das Ansteuern des Ventils mit dem Vorgang "Ankuppeln"
//    und das Absteuern des Ventils mit dem Vorgang "Abkuppeln".
//Bei Maschinen OHNE Kupplung am Rüstplatz wird die Funktion mit
//"I_SP_HYD_NEG_STOERUNG" gesteuert.
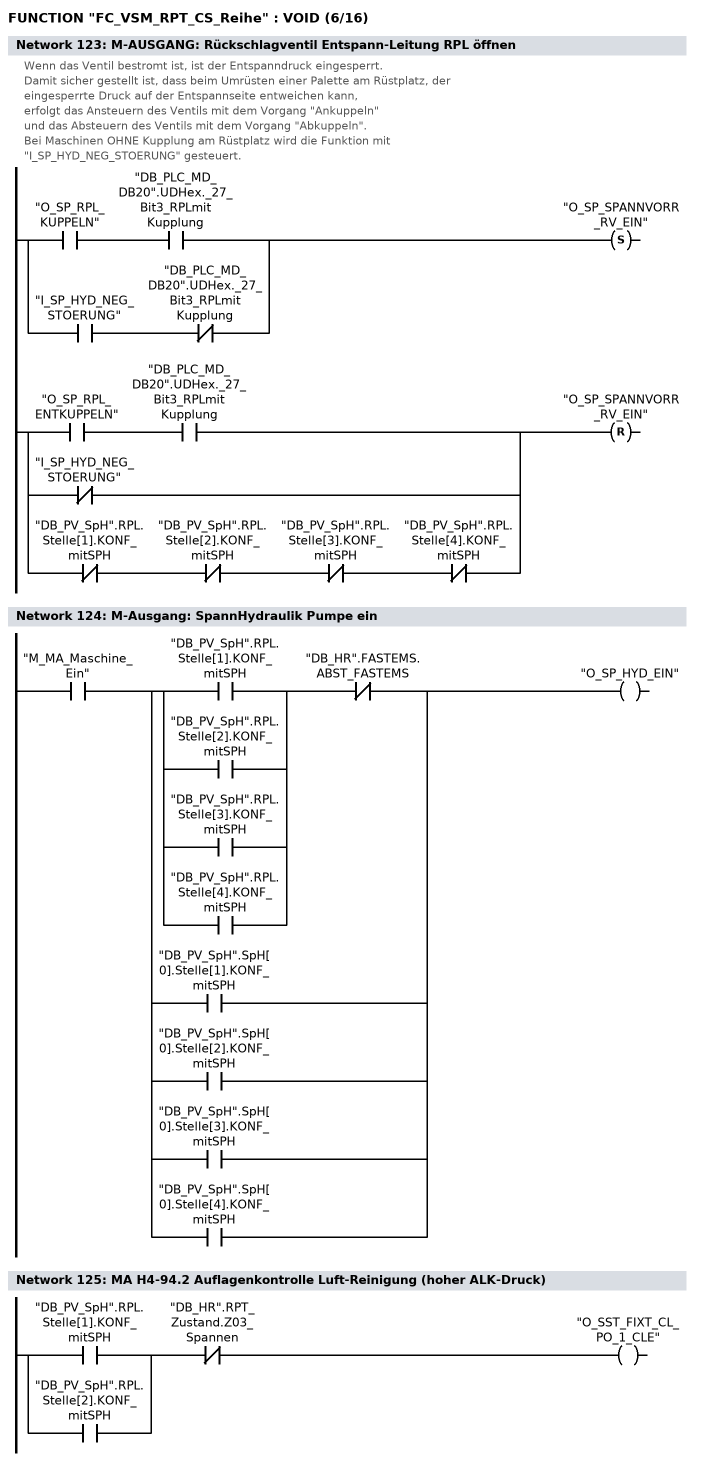
      U(    ;
      U     "O_SP_RPL_KUPPELN";
      U     "DB_PLC_MD_DB20".UDHex._27_Bit3_RPLmitKupplung;
      O     ;
      U     "I_SP_HYD_NEG_STOERUNG";
      UN    "DB_PLC_MD_DB20".UDHex._27_Bit3_RPLmitKupplung;
      )     ;
      S     "O_SP_SPANNVORR_RV_EIN";
      U(    ;
      U     "O_SP_RPL_ENTKUPPELN";
      U     "DB_PLC_MD_DB20".UDHex._27_Bit3_RPLmitKupplung;
      ON    "I_SP_HYD_NEG_STOERUNG";
      O     ;
      UN    "DB_PV_SpH".RPL.Stelle[1].KONF_mitSPH;
      UN    "DB_PV_SpH".RPL.Stelle[2].KONF_mitSPH;
      UN    "DB_PV_SpH".RPL.Stelle[3].KONF_mitSPH;
      UN    "DB_PV_SpH".RPL.Stelle[4].KONF_mitSPH;
      )     ;
      R     "O_SP_SPANNVORR_RV_EIN";
      NOP   0;
NETWORK
TITLE =M-Ausgang: SpannHydraulik Pumpe ein

      U     "M_MA_Maschine_Ein";
      U(    ;
      U(    ;
      O     "DB_PV_SpH".RPL.Stelle[1].KONF_mitSPH;
      O     "DB_PV_SpH".RPL.Stelle[2].KONF_mitSPH;
      O     "DB_PV_SpH".RPL.Stelle[3].KONF_mitSPH;
      O     "DB_PV_SpH".RPL.Stelle[4].KONF_mitSPH;
      )     ;
      UN    "DB_HR".FASTEMS.ABST_FASTEMS;
      O     "DB_PV_SpH".SpH[0].Stelle[1].KONF_mitSPH;
      O     "DB_PV_SpH".SpH[0].Stelle[2].KONF_mitSPH;
      O     "DB_PV_SpH".SpH[0].Stelle[3].KONF_mitSPH;
      O     "DB_PV_SpH".SpH[0].Stelle[4].KONF_mitSPH;
      )     ;
      =     "O_SP_HYD_EIN";
NETWORK
TITLE =MA H4-94.2 Auflagenkontrolle Luft-Reinigung (hoher ALK-Druck)

      U(    ;
      O     "DB_PV_SpH".RPL.Stelle[1].KONF_mitSPH;
      O     "DB_PV_SpH".RPL.Stelle[2].KONF_mitSPH;
      )     ;
      UN    "DB_HR".RPT_Zustand.Z03_Spannen;
      =     "O_SST_FIXT_CL_PO_1_CLE";
NETWORK
TITLE =Timer Laufzeit Auflagenkontrolle "Luft-Reinigung" entlüften
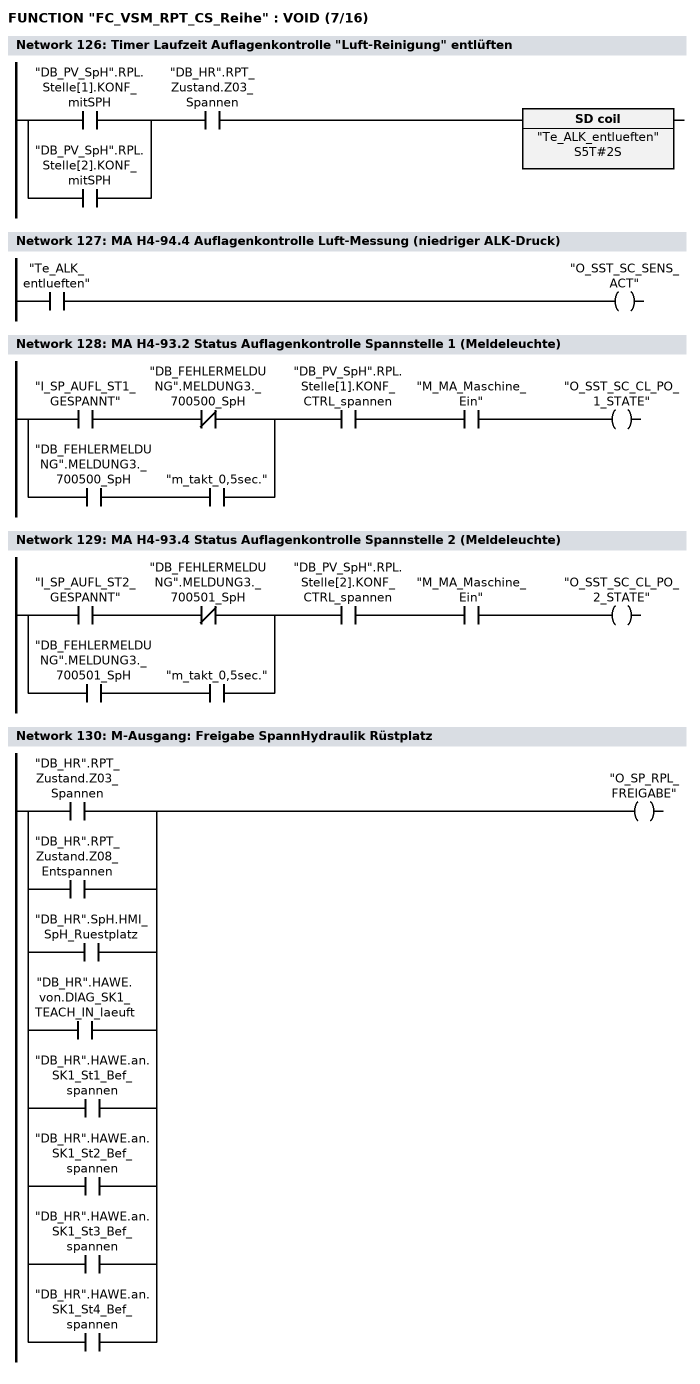

      U(    ;
      O     "DB_PV_SpH".RPL.Stelle[1].KONF_mitSPH;
      O     "DB_PV_SpH".RPL.Stelle[2].KONF_mitSPH;
      )     ;
      U     "DB_HR".RPT_Zustand.Z03_Spannen;
      L     S5T#2S;
      SE    "Te_ALK_entlueften";
NETWORK
TITLE =MA H4-94.4 Auflagenkontrolle Luft-Messung (niedriger ALK-Druck)

      U     "Te_ALK_entlueften";
      =     "O_SST_SC_SENS_ACT";
NETWORK
TITLE =MA H4-93.2 Status Auflagenkontrolle Spannstelle 1 (Meldeleuchte)

      U(    ;
      U     "I_SP_AUFL_ST1_GESPANNT";
      UN    "DB_FEHLERMELDUNG".MELDUNG3._700500_SpH;
      O     ;
      U     "DB_FEHLERMELDUNG".MELDUNG3._700500_SpH;
      U     "m_takt_0,5sec.";
      )     ;
      U     "DB_PV_SpH".RPL.Stelle[1].KONF_CTRL_spannen;
      U     "M_MA_Maschine_Ein";
      =     "O_SST_SC_CL_PO_1_STATE";
NETWORK
TITLE =MA H4-93.4 Status Auflagenkontrolle Spannstelle 2 (Meldeleuchte)

      U(    ;
      U     "I_SP_AUFL_ST2_GESPANNT";
      UN    "DB_FEHLERMELDUNG".MELDUNG3._700501_SpH;
      O     ;
      U     "DB_FEHLERMELDUNG".MELDUNG3._700501_SpH;
      U     "m_takt_0,5sec.";
      )     ;
      U     "DB_PV_SpH".RPL.Stelle[2].KONF_CTRL_spannen;
      U     "M_MA_Maschine_Ein";
      =     "O_SST_SC_CL_PO_2_STATE";
NETWORK
TITLE =M-Ausgang: Freigabe SpannHydraulik Rüstplatz

      O     "DB_HR".RPT_Zustand.Z03_Spannen;
      O     "DB_HR".RPT_Zustand.Z08_Entspannen;
      O     "DB_HR".SpH.HMI_SpH_Ruestplatz;
      O     "DB_HR".HAWE.von.DIAG_SK1_TEACH_IN_laeuft;
      O     "DB_HR".HAWE.an.SK1_St1_Bef_spannen;
      O     "DB_HR".HAWE.an.SK1_St2_Bef_spannen;
      O     "DB_HR".HAWE.an.SK1_St3_Bef_spannen;
      O     "DB_HR".HAWE.an.SK1_St4_Bef_spannen;
      =     "O_SP_RPL_FREIGABE";
NETWORK
TITLE =Anforderung an Rüstplatz-Achse: Auf PW-Wechsel-Position fahren
//In FC191 weiterverarbeitet.
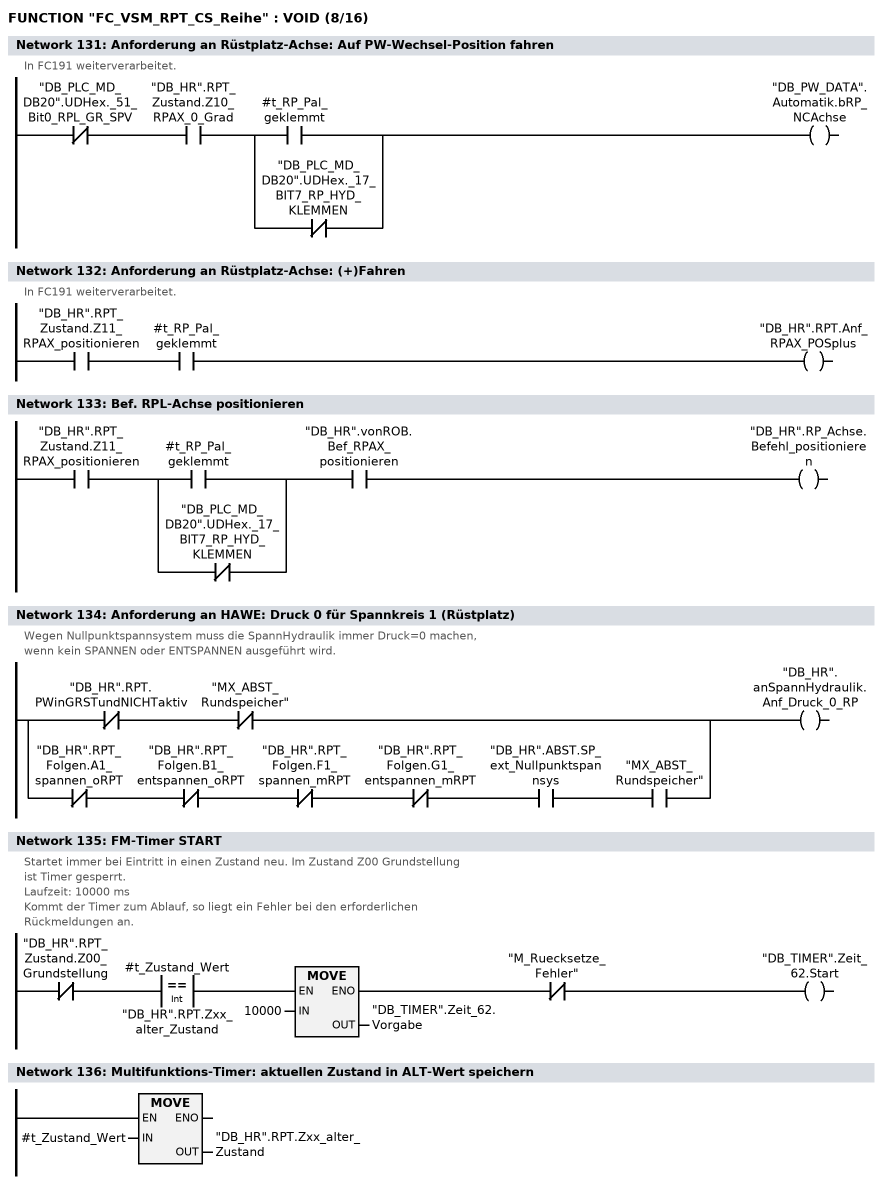
      UN    "DB_PLC_MD_DB20".UDHex._51_Bit0_RPL_GR_SPV;
      U     "DB_HR".RPT_Zustand.Z10_RPAX_0_Grad;
      U(    ;
      O     #t_RP_Pal_geklemmt;
      ON    "DB_PLC_MD_DB20".UDHex._17_BIT7_RP_HYD_KLEMMEN;
      )     ;
      =     "DB_PW_DATA".Automatik.bRP_NCAchse;
NETWORK
TITLE =Anforderung an Rüstplatz-Achse: (+)Fahren
//In FC191 weiterverarbeitet.
      U     "DB_HR".RPT_Zustand.Z11_RPAX_positionieren;
      U     #t_RP_Pal_geklemmt;
      =     "DB_HR".RPT.Anf_RPAX_POSplus;
NETWORK
TITLE =Bef. RPL-Achse positionieren

      U     "DB_HR".RPT_Zustand.Z11_RPAX_positionieren;
      U(    ;
      O     #t_RP_Pal_geklemmt;
      ON    "DB_PLC_MD_DB20".UDHex._17_BIT7_RP_HYD_KLEMMEN;
      )     ;
      U     "DB_HR".vonROB.Bef_RPAX_positionieren;
      =     "DB_HR".RP_Achse.Befehl_positionieren;
NETWORK
TITLE =Anforderung an HAWE: Druck 0 für Spannkreis 1 (Rüstplatz)
//Wegen Nullpunktspannsystem muss die SpannHydraulik immer Druck=0 machen,
//wenn kein SPANNEN oder ENTSPANNEN ausgeführt wird.
      UN    "DB_HR".RPT.PWinGRSTundNICHTaktiv;
      UN    "MX_ABST_Rundspeicher";
      O     ;
      UN    "DB_HR".RPT_Folgen.A1_spannen_oRPT;
      UN    "DB_HR".RPT_Folgen.B1_entspannen_oRPT;
      UN    "DB_HR".RPT_Folgen.F1_spannen_mRPT;
      UN    "DB_HR".RPT_Folgen.G1_entspannen_mRPT;
      U     "DB_HR".ABST.SP_ext_Nullpunktspannsys;
      U     "MX_ABST_Rundspeicher";
      =     "DB_HR".anSpannHydraulik.Anf_Druck_0_RP;
NETWORK
TITLE =FM-Timer START
//Startet immer bei Eintritt in einen Zustand neu. Im Zustand Z00 Grundstellung
//ist Timer gesperrt.
//Laufzeit: 10000 ms
//Kommt der Timer zum Ablauf, so liegt ein Fehler bei den erforderlichen
//Rückmeldungen an.
      U(    ;
      UN    "DB_HR".RPT_Zustand.Z00_Grundstellung;
      U(    ;
      L     #t_Zustand_Wert;
      L     "DB_HR".RPT.Zxx_alter_Zustand;
      ==I   ;
      )     ;
      SPBNB _028;
      L     10000;
      T     "DB_TIMER".Zeit_62.Vorgabe;
      SET   ;
      SAVE  ;
      CLR   ;
_028: U     BIE;
      )     ;
      UN    "M_Ruecksetze_Fehler";
      =     "DB_TIMER".Zeit_62.Start;
NETWORK
TITLE =Multifunktions-Timer: aktuellen Zustand in ALT-Wert speichern

      L     #t_Zustand_Wert;
      T     "DB_HR".RPT.Zxx_alter_Zustand;
      NOP   0;
NETWORK
TITLE =700455 Rüstplatz: Meldung Palette geklemmt fehlt!
//      U     "DB_HR".RPT_Zustand.Z01_PalKlemmung_ein
//      UN    #t_RP_Pal_geklemmt
//      U     "DB_PLC_MD_DB20".UDHex._17_BIT7_RP_HYD_KLEMMEN
//      U     "DB_TIMER".Zeit_62.Ausgang
//      =     "DB_FEHLERMELDUNG".MELDUNG3._700455_RPT
//
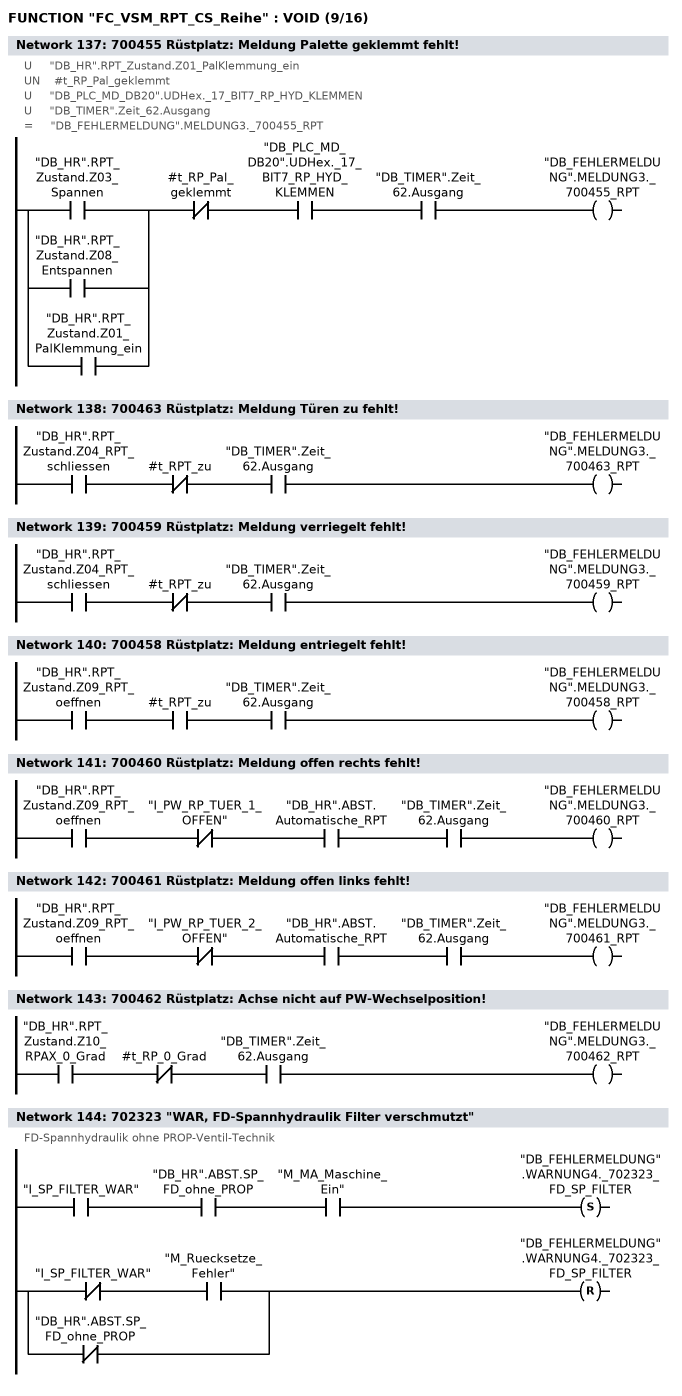
      U(    ;
      O     "DB_HR".RPT_Zustand.Z03_Spannen;
      O     "DB_HR".RPT_Zustand.Z08_Entspannen;
      O     "DB_HR".RPT_Zustand.Z01_PalKlemmung_ein;
      )     ;
      UN    #t_RP_Pal_geklemmt;
      U     "DB_PLC_MD_DB20".UDHex._17_BIT7_RP_HYD_KLEMMEN;
      U     "DB_TIMER".Zeit_62.Ausgang;
      =     "DB_FEHLERMELDUNG".MELDUNG3._700455_RPT;
NETWORK
TITLE =700463 Rüstplatz: Meldung Türen zu fehlt!

      U     "DB_HR".RPT_Zustand.Z04_RPT_schliessen;
      UN    #t_RPT_zu;
      U     "DB_TIMER".Zeit_62.Ausgang;
      =     "DB_FEHLERMELDUNG".MELDUNG3._700463_RPT;
NETWORK
TITLE =700459 Rüstplatz: Meldung verriegelt fehlt!

      U     "DB_HR".RPT_Zustand.Z04_RPT_schliessen;
      UN    #t_RPT_zu;
      U     "DB_TIMER".Zeit_62.Ausgang;
      =     "DB_FEHLERMELDUNG".MELDUNG3._700459_RPT;
NETWORK
TITLE =700458 Rüstplatz: Meldung entriegelt fehlt!

      U     "DB_HR".RPT_Zustand.Z09_RPT_oeffnen;
      U     #t_RPT_zu;
      U     "DB_TIMER".Zeit_62.Ausgang;
      =     "DB_FEHLERMELDUNG".MELDUNG3._700458_RPT;
NETWORK
TITLE =700460 Rüstplatz: Meldung offen rechts fehlt!

      U     "DB_HR".RPT_Zustand.Z09_RPT_oeffnen;
      UN    "I_PW_RP_TUER_1_OFFEN";
      U     "DB_HR".ABST.Automatische_RPT;
      U     "DB_TIMER".Zeit_62.Ausgang;
      =     "DB_FEHLERMELDUNG".MELDUNG3._700460_RPT;
NETWORK
TITLE =700461 Rüstplatz: Meldung offen links fehlt!

      U     "DB_HR".RPT_Zustand.Z09_RPT_oeffnen;
      UN    "I_PW_RP_TUER_2_OFFEN";
      U     "DB_HR".ABST.Automatische_RPT;
      U     "DB_TIMER".Zeit_62.Ausgang;
      =     "DB_FEHLERMELDUNG".MELDUNG3._700461_RPT;
NETWORK
TITLE =700462 Rüstplatz: Achse nicht auf PW-Wechselposition!

      U     "DB_HR".RPT_Zustand.Z10_RPAX_0_Grad;
      UN    #t_RP_0_Grad;
      U     "DB_TIMER".Zeit_62.Ausgang;
      =     "DB_FEHLERMELDUNG".MELDUNG3._700462_RPT;
NETWORK
TITLE =702323 "WAR, FD-Spannhydraulik Filter verschmutzt"
//FD-Spannhydraulik ohne PROP-Ventil-Technik
      U     "I_SP_FILTER_WAR";
      U     "DB_HR".ABST.SP_FD_ohne_PROP;
      U     "M_MA_Maschine_Ein";
      S     "DB_FEHLERMELDUNG".WARNUNG4._702323_FD_SP_FILTER;
      U(    ;
      UN    "I_SP_FILTER_WAR";
      U     "M_Ruecksetze_Fehler";
      ON    "DB_HR".ABST.SP_FD_ohne_PROP;
      )     ;
      R     "DB_FEHLERMELDUNG".WARNUNG4._702323_FD_SP_FILTER;
      NOP   0;
NETWORK
TITLE =FD-Spannhydraulik OHNE PROP: max Fehlerlaufzeit bis VS-HLT
//Konfiguartionswert in Millisekunden wandeln
//Init: 20000 ms
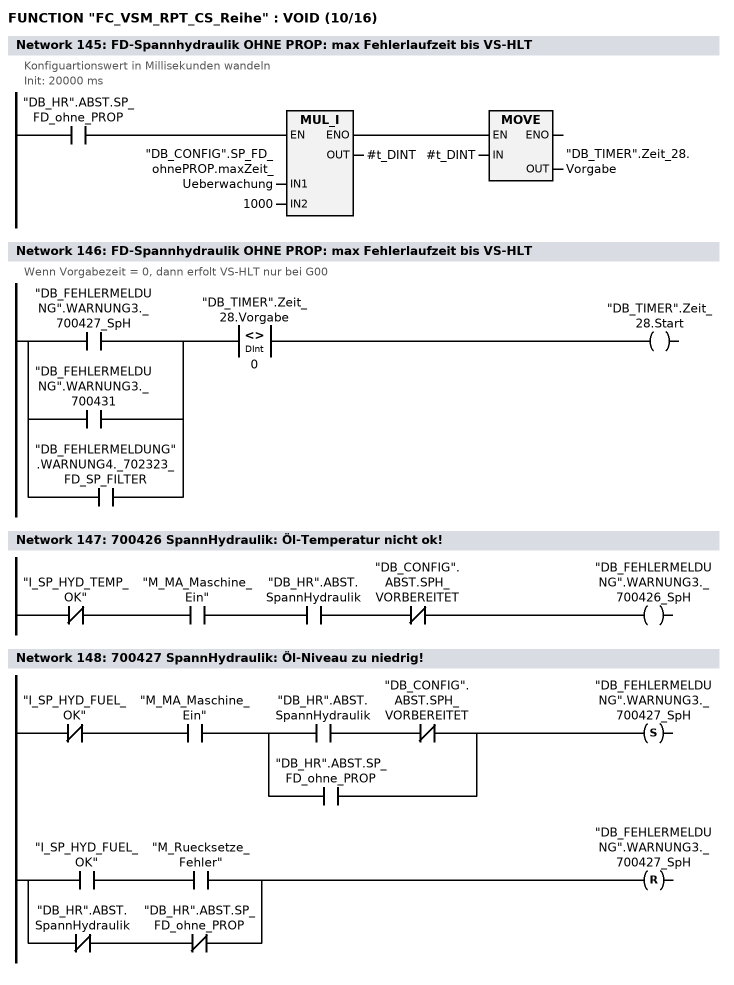
      U(    ;
      U     "DB_HR".ABST.SP_FD_ohne_PROP;
      SPBNB _029;
      L     "DB_CONFIG".SP_FD_ohnePROP.maxZeit_Ueberwachung;
      L     1000;
      *I    ;
      T     #t_DINT;
      UN    OV;
      SAVE  ;
      CLR   ;
_029: U     BIE;
      )     ;
      SPBNB _02a;
      L     #t_DINT;
      T     "DB_TIMER".Zeit_28.Vorgabe;
_02a: NOP   0;
NETWORK
TITLE =FD-Spannhydraulik OHNE PROP: max Fehlerlaufzeit bis VS-HLT
//Wenn Vorgabezeit = 0, dann erfolt VS-HLT nur bei G00
      U(    ;
      O     "DB_FEHLERMELDUNG".WARNUNG3._700427_SpH;
      O     "DB_FEHLERMELDUNG".WARNUNG3._700431;
      O     "DB_FEHLERMELDUNG".WARNUNG4._702323_FD_SP_FILTER;
      )     ;
      U(    ;
      L     "DB_TIMER".Zeit_28.Vorgabe;
      L     0;
      <>D   ;
      )     ;
      =     "DB_TIMER".Zeit_28.Start;
NETWORK
TITLE =700426 SpannHydraulik: Öl-Temperatur nicht ok!

      UN    "I_SP_HYD_TEMP_OK";
      U     "M_MA_Maschine_Ein";
      U     "DB_HR".ABST.SpannHydraulik;
      UN    "DB_CONFIG".ABST.SPH_VORBEREITET;
      =     "DB_FEHLERMELDUNG".WARNUNG3._700426_SpH;
NETWORK
TITLE =700427 SpannHydraulik: Öl-Niveau zu niedrig!

      UN    "I_SP_HYD_FUEL_OK";
      U     "M_MA_Maschine_Ein";
      U(    ;
      U     "DB_HR".ABST.SpannHydraulik;
      UN    "DB_CONFIG".ABST.SPH_VORBEREITET;
      O     "DB_HR".ABST.SP_FD_ohne_PROP;
      )     ;
      S     "DB_FEHLERMELDUNG".WARNUNG3._700427_SpH;
      U(    ;
      U     "I_SP_HYD_FUEL_OK";
      U     "M_Ruecksetze_Fehler";
      O     ;
      UN    "DB_HR".ABST.SpannHydraulik;
      UN    "DB_HR".ABST.SP_FD_ohne_PROP;
      )     ;
      R     "DB_FEHLERMELDUNG".WARNUNG3._700427_SpH;
      NOP   0;
NETWORK
TITLE =700209 "SPI-VS-H, Spannhydraulik Überwachung Füllstand / Tempera
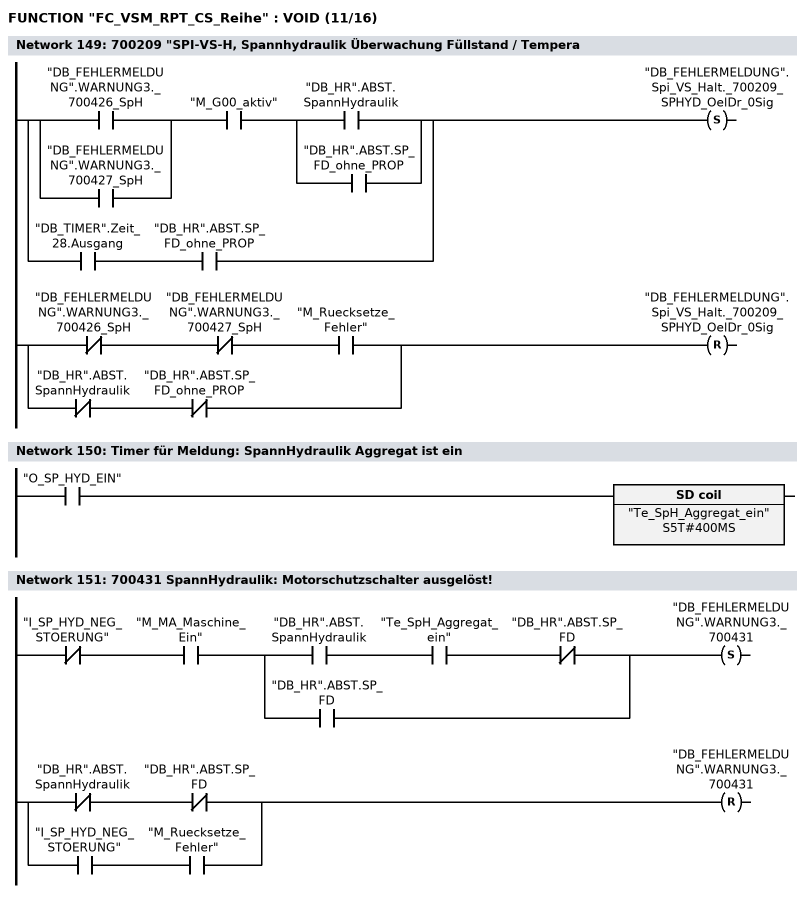

      U(    ;
      U(    ;
      O     "DB_FEHLERMELDUNG".WARNUNG3._700426_SpH;
      O     "DB_FEHLERMELDUNG".WARNUNG3._700427_SpH;
      )     ;
      U     "M_G00_aktiv";
      U(    ;
      O     "DB_HR".ABST.SpannHydraulik;
      O     "DB_HR".ABST.SP_FD_ohne_PROP;
      )     ;
      O     ;
      U     "DB_TIMER".Zeit_28.Ausgang;
      U     "DB_HR".ABST.SP_FD_ohne_PROP;
      )     ;
      S     "DB_FEHLERMELDUNG".Spi_VS_Halt._700209_SPHYD_OelDr_0Sig;
      U(    ;
      UN    "DB_FEHLERMELDUNG".WARNUNG3._700426_SpH;
      UN    "DB_FEHLERMELDUNG".WARNUNG3._700427_SpH;
      U     "M_Ruecksetze_Fehler";
      O     ;
      UN    "DB_HR".ABST.SpannHydraulik;
      UN    "DB_HR".ABST.SP_FD_ohne_PROP;
      )     ;
      R     "DB_FEHLERMELDUNG".Spi_VS_Halt._700209_SPHYD_OelDr_0Sig;
      NOP   0;
NETWORK
TITLE =Timer für Meldung: SpannHydraulik Aggregat ist ein

      U     "O_SP_HYD_EIN";
      L     S5T#400MS;
      SE    "Te_SpH_Aggregat_ein";
NETWORK
TITLE =700431 SpannHydraulik: Motorschutzschalter ausgelöst!

      UN    "I_SP_HYD_NEG_STOERUNG";
      U     "M_MA_Maschine_Ein";
      U(    ;
      U     "DB_HR".ABST.SpannHydraulik;
      U     "Te_SpH_Aggregat_ein";
      UN    "DB_HR".ABST.SP_FD;
      O     "DB_HR".ABST.SP_FD;
      )     ;
      S     "DB_FEHLERMELDUNG".WARNUNG3._700431;
      U(    ;
      UN    "DB_HR".ABST.SpannHydraulik;
      UN    "DB_HR".ABST.SP_FD;
      O     ;
      U     "I_SP_HYD_NEG_STOERUNG";
      U     "M_Ruecksetze_Fehler";
      )     ;
      R     "DB_FEHLERMELDUNG".WARNUNG3._700431;
      NOP   0;
NETWORK
TITLE =700452 SpannHydraulik: Rüstplatz Spannstelle 1 nicht gespannt!
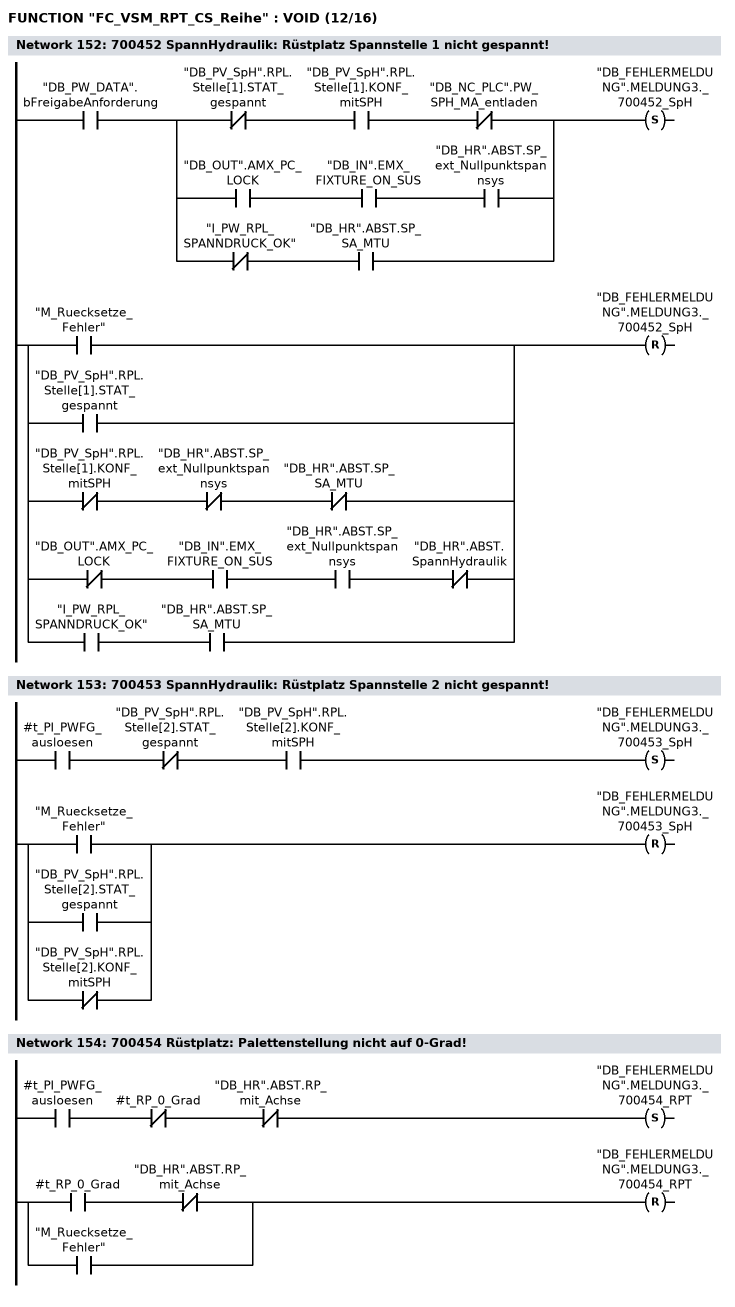

      U     "DB_PW_DATA".bFreigabeAnforderung;
      U(    ;
      UN    "DB_PV_SpH".RPL.Stelle[1].STAT_gespannt;
      U     "DB_PV_SpH".RPL.Stelle[1].KONF_mitSPH;
      UN    "DB_NC_PLC".PW_SPH_MA_entladen;
      O     ;
      U     "DB_OUT".AMX_PC_LOCK;
      U     "DB_IN".EMX_FIXTURE_ON_SUS;
      U     "DB_HR".ABST.SP_ext_Nullpunktspannsys;
      O     ;
      UN    "I_PW_RPL_SPANNDRUCK_OK";
      U     "DB_HR".ABST.SP_SA_MTU;
      )     ;
      S     "DB_FEHLERMELDUNG".MELDUNG3._700452_SpH;
      U(    ;
      O     "M_Ruecksetze_Fehler";
      O     "DB_PV_SpH".RPL.Stelle[1].STAT_gespannt;
      O     ;
      UN    "DB_PV_SpH".RPL.Stelle[1].KONF_mitSPH;
      UN    "DB_HR".ABST.SP_ext_Nullpunktspannsys;
      UN    "DB_HR".ABST.SP_SA_MTU;
      O     ;
      UN    "DB_OUT".AMX_PC_LOCK;
      U     "DB_IN".EMX_FIXTURE_ON_SUS;
      U     "DB_HR".ABST.SP_ext_Nullpunktspannsys;
      UN    "DB_HR".ABST.SpannHydraulik;
      O     ;
      U     "I_PW_RPL_SPANNDRUCK_OK";
      U     "DB_HR".ABST.SP_SA_MTU;
      )     ;
      R     "DB_FEHLERMELDUNG".MELDUNG3._700452_SpH;
      NOP   0;
NETWORK
TITLE =700453 SpannHydraulik: Rüstplatz Spannstelle 2 nicht gespannt!

      U     #t_PI_PWFG_ausloesen;
      UN    "DB_PV_SpH".RPL.Stelle[2].STAT_gespannt;
      U     "DB_PV_SpH".RPL.Stelle[2].KONF_mitSPH;
      S     "DB_FEHLERMELDUNG".MELDUNG3._700453_SpH;
      U(    ;
      O     "M_Ruecksetze_Fehler";
      O     "DB_PV_SpH".RPL.Stelle[2].STAT_gespannt;
      ON    "DB_PV_SpH".RPL.Stelle[2].KONF_mitSPH;
      )     ;
      R     "DB_FEHLERMELDUNG".MELDUNG3._700453_SpH;
      NOP   0;
NETWORK
TITLE =700454 Rüstplatz: Palettenstellung nicht auf 0-Grad!

      U     #t_PI_PWFG_ausloesen;
      UN    #t_RP_0_Grad;
      UN    "DB_HR".ABST.RP_mit_Achse;
      S     "DB_FEHLERMELDUNG".MELDUNG3._700454_RPT;
      U(    ;
      U     #t_RP_0_Grad;
      UN    "DB_HR".ABST.RP_mit_Achse;
      O     "M_Ruecksetze_Fehler";
      )     ;
      R     "DB_FEHLERMELDUNG".MELDUNG3._700454_RPT;
      NOP   0;
NETWORK
TITLE =702412 "Meldung, keine PW-Freigabe; SOKO fordert ankuppeln"
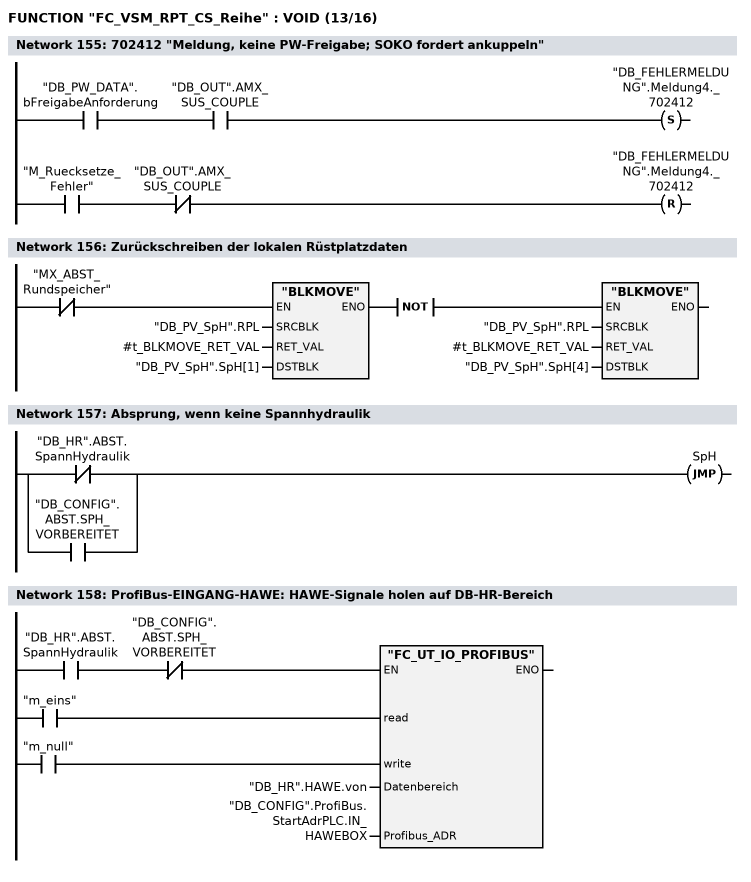

      U     "DB_PW_DATA".bFreigabeAnforderung;
      U     "DB_OUT".AMX_SUS_COUPLE;
      S     "DB_FEHLERMELDUNG".Meldung4._702412;
      U     "M_Ruecksetze_Fehler";
      UN    "DB_OUT".AMX_SUS_COUPLE;
      R     "DB_FEHLERMELDUNG".Meldung4._702412;
      NOP   0;
NETWORK
TITLE =Zurückschreiben der lokalen Rüstplatzdaten

      U(    ;
      UN    "MX_ABST_Rundspeicher";
      SPBNB _02b;
      CALL "BLKMOVE" (
           SRCBLK                   := "DB_PV_SpH".RPL,
           RET_VAL                  := #t_BLKMOVE_RET_VAL,
           DSTBLK                   := "DB_PV_SpH".SpH[1]);
_02b: U     BIE;
      )     ;
      NOT   ;
      SPBNB _02c;
      CALL "BLKMOVE" (
           SRCBLK                   := "DB_PV_SpH".RPL,
           RET_VAL                  := #t_BLKMOVE_RET_VAL,
           DSTBLK                   := "DB_PV_SpH".SpH[4]);
_02c: NOP   0;
NETWORK
TITLE =Absprung, wenn keine Spannhydraulik

      ON    "DB_HR".ABST.SpannHydraulik;
      O     "DB_CONFIG".ABST.SPH_VORBEREITET;
      SPB   SpH;
NETWORK
TITLE =ProfiBus-EINGANG-HAWE: HAWE-Signale holen auf DB-HR-Bereich

      U     "m_eins";
      =     L     21.0;
      BLD   103;
      U     "m_null";
      =     L     21.1;
      BLD   103;
      U     "DB_HR".ABST.SpannHydraulik;
      UN    "DB_CONFIG".ABST.SPH_VORBEREITET;
      SPBNB _02d;
      CALL "FC_UT_IO_PROFIBUS" (
           read                     := L     21.0,
           write                    := L     21.1,
           Datenbereich             := "DB_HR".HAWE.von,
           Profibus_ADR             := "DB_CONFIG".ProfiBus.StartAdrPLC.IN_HAWEBOX);
_02d: NOP   0;
NETWORK
TITLE =>>>>> FB_SPH: Aufruf SpannHydraulik OHNE FD
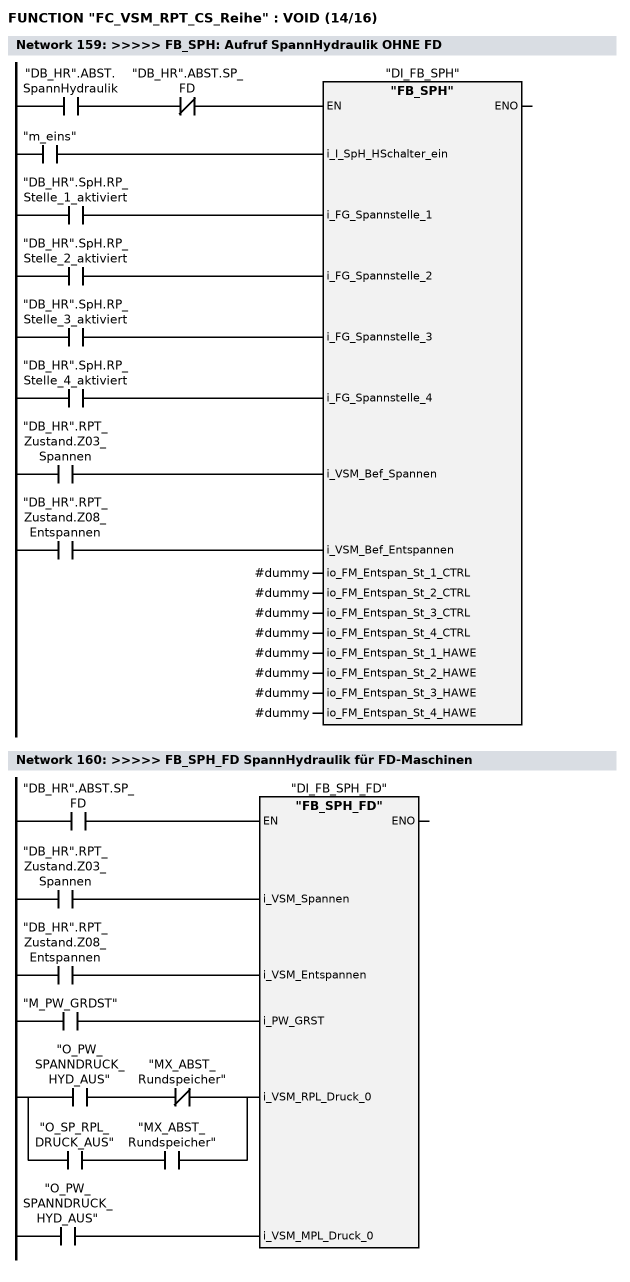

      U     "m_eins";
      =     L     21.0;
      BLD   103;
      U     "DB_HR".SpH.RP_Stelle_1_aktiviert;
      =     L     21.1;
      BLD   103;
      U     "DB_HR".SpH.RP_Stelle_2_aktiviert;
      =     L     21.2;
      BLD   103;
      U     "DB_HR".SpH.RP_Stelle_3_aktiviert;
      =     L     21.3;
      BLD   103;
      U     "DB_HR".SpH.RP_Stelle_4_aktiviert;
      =     L     21.4;
      BLD   103;
      U     "DB_HR".RPT_Zustand.Z03_Spannen;
      =     L     21.5;
      BLD   103;
      U     "DB_HR".RPT_Zustand.Z08_Entspannen;
      =     L     21.6;
      BLD   103;
      U     "DB_HR".ABST.SpannHydraulik;
      UN    "DB_HR".ABST.SP_FD;
      SPBNB _02e;
      CALL "FB_SPH" , "DI_FB_SPH" (
           i_I_SpH_HSchalter_ein    := L     21.0,
           i_FG_Spannstelle_1       := L     21.1,
           i_FG_Spannstelle_2       := L     21.2,
           i_FG_Spannstelle_3       := L     21.3,
           i_FG_Spannstelle_4       := L     21.4,
           i_VSM_Bef_Spannen        := L     21.5,
           i_VSM_Bef_Entspannen     := L     21.6,
           io_FM_Entspan_St_1_CTRL  := #dummy,
           io_FM_Entspan_St_2_CTRL  := #dummy,
           io_FM_Entspan_St_3_CTRL  := #dummy,
           io_FM_Entspan_St_4_CTRL  := #dummy,
           io_FM_Entspan_St_1_HAWE  := #dummy,
           io_FM_Entspan_St_2_HAWE  := #dummy,
           io_FM_Entspan_St_3_HAWE  := #dummy,
           io_FM_Entspan_St_4_HAWE  := #dummy);

_02e: NOP   0;
NETWORK
TITLE =>>>>> FB_SPH_FD SpannHydraulik für FD-Maschinen

      U     "DB_HR".RPT_Zustand.Z03_Spannen;
      =     L     21.0;
      BLD   103;
      U     "DB_HR".RPT_Zustand.Z08_Entspannen;
      =     L     21.1;
      BLD   103;
      U     "M_PW_GRDST";
      =     L     21.2;
      BLD   103;
      U(    ;
      U     "O_PW_SPANNDRUCK_HYD_AUS";
      UN    "MX_ABST_Rundspeicher";
      O     ;
      U     "O_SP_RPL_DRUCK_AUS";
      U     "MX_ABST_Rundspeicher";
      )     ;
      =     L     21.3;
      BLD   103;
      U     "O_PW_SPANNDRUCK_HYD_AUS";
      =     L     21.4;
      BLD   103;
      U     "DB_HR".ABST.SP_FD;
      SPBNB _02f;
      CALL "FB_SPH_FD" , "DI_FB_SPH_FD" (
           i_VSM_Spannen            := L     21.0,
           i_VSM_Entspannen         := L     21.1,
           i_PW_GRST                := L     21.2,
           i_VSM_RPL_Druck_0        := L     21.3,
           i_VSM_MPL_Druck_0        := L     21.4);
_02f: NOP   0;
NETWORK
TITLE =ProfiBus-AUSGANG-HAWE: DB_HR-Bereich an HAWE senden
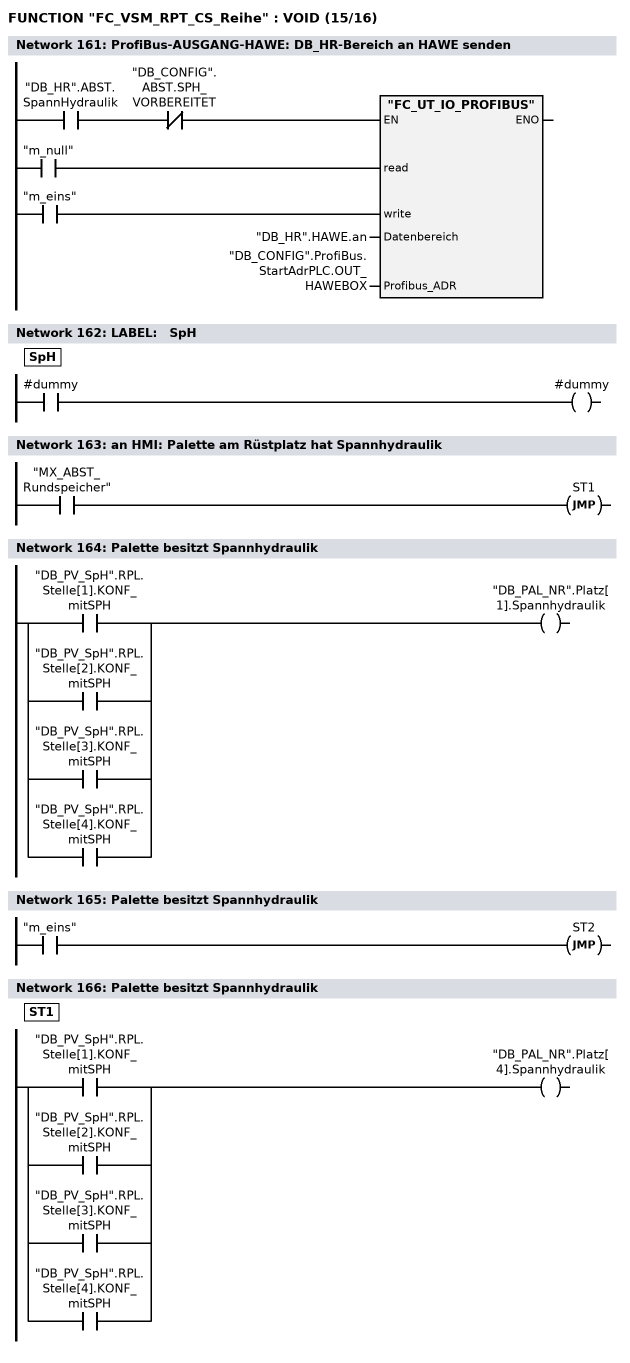

      U     "m_null";
      =     L     21.0;
      BLD   103;
      U     "m_eins";
      =     L     21.1;
      BLD   103;
      U     "DB_HR".ABST.SpannHydraulik;
      UN    "DB_CONFIG".ABST.SPH_VORBEREITET;
      SPBNB _030;
      CALL "FC_UT_IO_PROFIBUS" (
           read                     := L     21.0,
           write                    := L     21.1,
           Datenbereich             := "DB_HR".HAWE.an,
           Profibus_ADR             := "DB_CONFIG".ProfiBus.StartAdrPLC.OUT_HAWEBOX);
_030: NOP   0;
NETWORK
TITLE =LABEL:   SpH

SpH:  U     #dummy;
      =     #dummy;
NETWORK
TITLE =an HMI: Palette am Rüstplatz hat Spannhydraulik

      U     "MX_ABST_Rundspeicher";
      SPB   ST1;
NETWORK
TITLE =Palette besitzt Spannhydraulik

      O     "DB_PV_SpH".RPL.Stelle[1].KONF_mitSPH;
      O     "DB_PV_SpH".RPL.Stelle[2].KONF_mitSPH;
      O     "DB_PV_SpH".RPL.Stelle[3].KONF_mitSPH;
      O     "DB_PV_SpH".RPL.Stelle[4].KONF_mitSPH;
      =     "DB_PAL_NR".Platz[1].Spannhydraulik;
NETWORK
TITLE =Palette besitzt Spannhydraulik

      U     "m_eins";
      SPB   ST2;
NETWORK
TITLE =Palette besitzt Spannhydraulik

ST1:  O     "DB_PV_SpH".RPL.Stelle[1].KONF_mitSPH;
      O     "DB_PV_SpH".RPL.Stelle[2].KONF_mitSPH;
      O     "DB_PV_SpH".RPL.Stelle[3].KONF_mitSPH;
      O     "DB_PV_SpH".RPL.Stelle[4].KONF_mitSPH;
      =     "DB_PAL_NR".Platz[4].Spannhydraulik;
NETWORK
TITLE =M-Ausgang: SpannHydraulik Rüstplatz entkuppeln
//ABST: "SpannHydraulik vorbereitet":
//Kupplung für RP und MA abkuppeln fest auf "1" sein
//Kupplung für RP und MA ankuppeln fest auf "0" sein
//
//ABST: ext.Nullpunktspannsystem:
//Kupplung am RP mit pos.Flanke "PW_in_GRST" ankuppeln
//Kupplung am Rüstplatz mit "Taste PW-Freigabe" abkuppeln
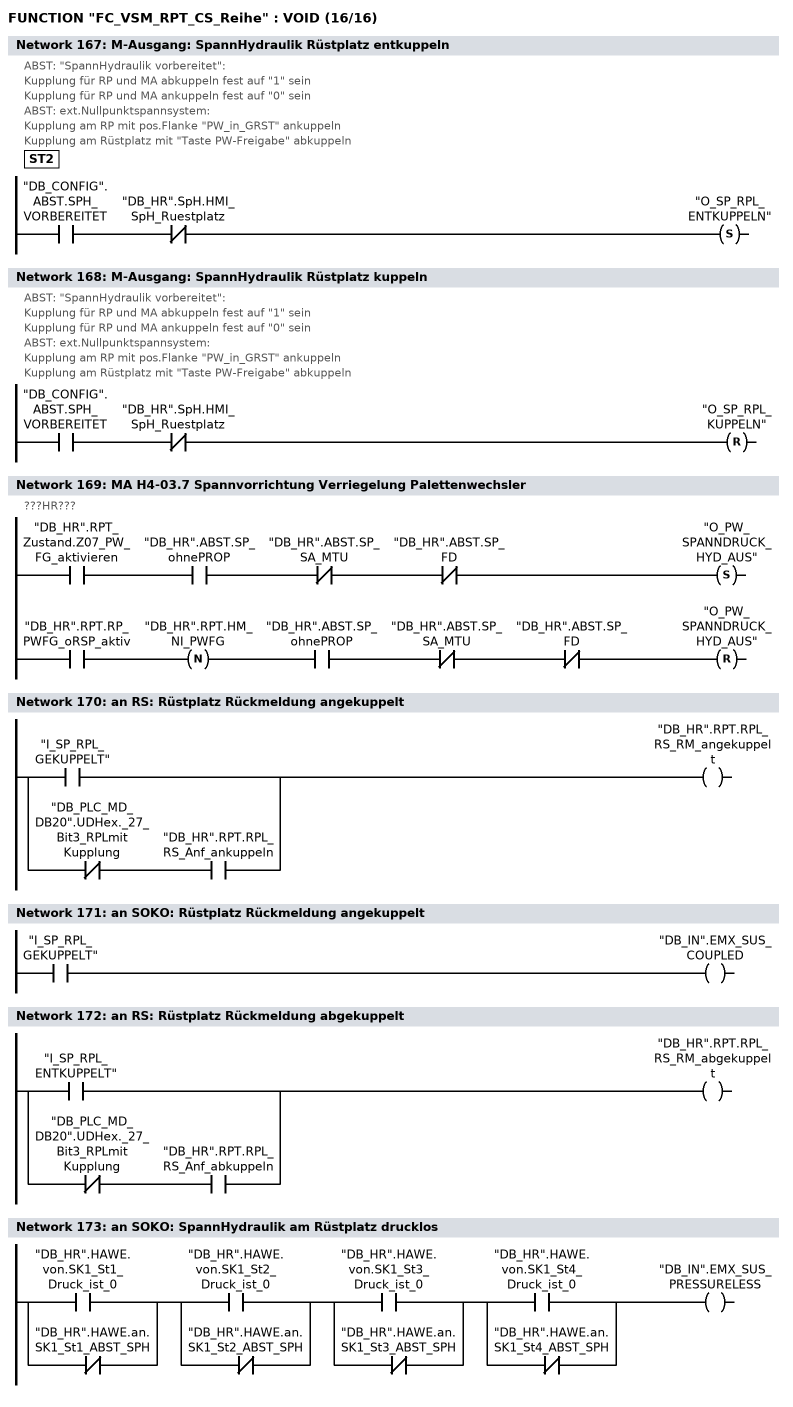
ST2:  U     "DB_CONFIG".ABST.SPH_VORBEREITET;
      UN    "DB_HR".SpH.HMI_SpH_Ruestplatz;
      S     "O_SP_RPL_ENTKUPPELN";
NETWORK
TITLE =M-Ausgang: SpannHydraulik Rüstplatz kuppeln
//ABST: "SpannHydraulik vorbereitet":
//Kupplung für RP und MA abkuppeln fest auf "1" sein
//Kupplung für RP und MA ankuppeln fest auf "0" sein
//
//ABST: ext.Nullpunktspannsystem:
//Kupplung am RP mit pos.Flanke "PW_in_GRST" ankuppeln
//Kupplung am Rüstplatz mit "Taste PW-Freigabe" abkuppeln
      U     "DB_CONFIG".ABST.SPH_VORBEREITET;
      UN    "DB_HR".SpH.HMI_SpH_Ruestplatz;
      R     "O_SP_RPL_KUPPELN";
NETWORK
TITLE =MA H4-03.7 Spannvorrichtung Verriegelung Palettenwechsler
//???HR???
      U     "DB_HR".RPT_Zustand.Z07_PW_FG_aktivieren;
      U     "DB_HR".ABST.SP_ohnePROP;
      UN    "DB_HR".ABST.SP_SA_MTU;
      UN    "DB_HR".ABST.SP_FD;
      S     "O_PW_SPANNDRUCK_HYD_AUS";
      U     "DB_HR".RPT.RP_PWFG_oRSP_aktiv;
      FN    "DB_HR".RPT.HM_NI_PWFG;
      U     "DB_HR".ABST.SP_ohnePROP;
      UN    "DB_HR".ABST.SP_SA_MTU;
      UN    "DB_HR".ABST.SP_FD;
      R     "O_PW_SPANNDRUCK_HYD_AUS";
      NOP   0;
NETWORK
TITLE =an RS: Rüstplatz Rückmeldung angekuppelt

      O     "I_SP_RPL_GEKUPPELT";
      O     ;
      UN    "DB_PLC_MD_DB20".UDHex._27_Bit3_RPLmitKupplung;
      U     "DB_HR".RPT.RPL_RS_Anf_ankuppeln;
      =     "DB_HR".RPT.RPL_RS_RM_angekuppelt;
NETWORK
TITLE =an SOKO: Rüstplatz Rückmeldung angekuppelt

      U     "I_SP_RPL_GEKUPPELT";
      =     "DB_IN".EMX_SUS_COUPLED;
NETWORK
TITLE =an RS: Rüstplatz Rückmeldung abgekuppelt

      O     "I_SP_RPL_ENTKUPPELT";
      O     ;
      UN    "DB_PLC_MD_DB20".UDHex._27_Bit3_RPLmitKupplung;
      U     "DB_HR".RPT.RPL_RS_Anf_abkuppeln;
      =     "DB_HR".RPT.RPL_RS_RM_abgekuppelt;
NETWORK
TITLE =an SOKO: SpannHydraulik am Rüstplatz drucklos

      U(    ;
      O     "DB_HR".HAWE.von.SK1_St1_Druck_ist_0;
      ON    "DB_HR".HAWE.an.SK1_St1_ABST_SPH;
      )     ;
      U(    ;
      O     "DB_HR".HAWE.von.SK1_St2_Druck_ist_0;
      ON    "DB_HR".HAWE.an.SK1_St2_ABST_SPH;
      )     ;
      U(    ;
      O     "DB_HR".HAWE.von.SK1_St3_Druck_ist_0;
      ON    "DB_HR".HAWE.an.SK1_St3_ABST_SPH;
      )     ;
      U(    ;
      O     "DB_HR".HAWE.von.SK1_St4_Druck_ist_0;
      ON    "DB_HR".HAWE.an.SK1_St4_ABST_SPH;
      )     ;
      =     "DB_IN".EMX_SUS_PRESSURELESS;
NETWORK
TITLE ================= SpH für Maschine OHNE PW ======================

      UN    "DB_HR".ABST.SP_ohnePW_OFFEN_Tuer;
      UN    "DB_HR".ABST.SP_ohnePW_ZU_Tuer;
      SPB   RPT;
SpH2: NOP   0;

NETWORK
TITLE =ProfiBus-EINGANG-HAWE: HAWE-Signale holen auf DB-HR-Bereich
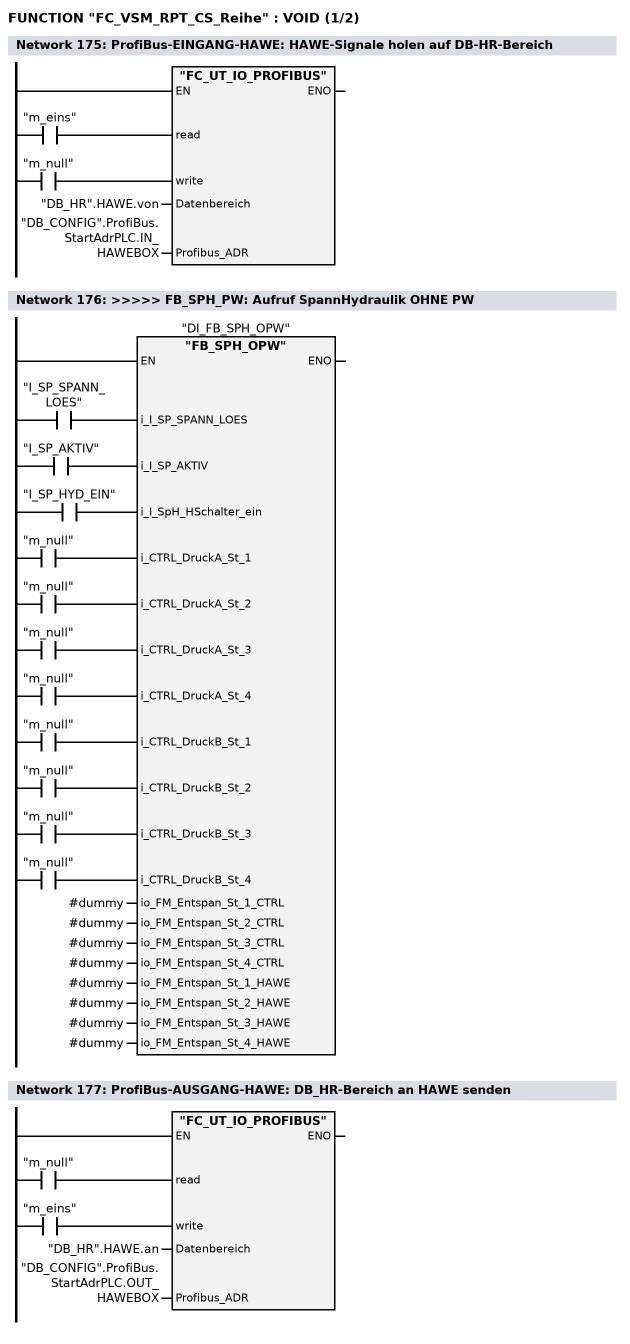

      U     "m_eins";
      =     L     21.0;
      BLD   103;
      U     "m_null";
      =     L     21.1;
      BLD   103;
      CALL "FC_UT_IO_PROFIBUS" (
           read                     := L     21.0,
           write                    := L     21.1,
           Datenbereich             := "DB_HR".HAWE.von,
           Profibus_ADR             := "DB_CONFIG".ProfiBus.StartAdrPLC.IN_HAWEBOX);
      NOP   0;
NETWORK
TITLE =>>>>> FB_SPH_PW: Aufruf SpannHydraulik OHNE PW

      U     "I_SP_SPANN_LOES";
      =     L     21.0;
      BLD   103;
      U     "I_SP_AKTIV";
      =     L     21.1;
      BLD   103;
      U     "I_SP_HYD_EIN";
      =     L     21.2;
      BLD   103;
      U     "m_null";
      =     L     21.3;
      BLD   103;
      U     "m_null";
      =     L     21.4;
      BLD   103;
      U     "m_null";
      =     L     21.5;
      BLD   103;
      U     "m_null";
      =     L     21.6;
      BLD   103;
      U     "m_null";
      =     L     21.7;
      BLD   103;
      U     "m_null";
      =     L     22.0;
      BLD   103;
      U     "m_null";
      =     L     22.1;
      BLD   103;
      U     "m_null";
      =     L     22.2;
      BLD   103;
      CALL "FB_SPH_OPW" , "DI_FB_SPH_OPW" (
           i_I_SP_SPANN_LOES        := L     21.0,
           i_I_SP_AKTIV             := L     21.1,
           i_I_SpH_HSchalter_ein    := L     21.2,
           i_CTRL_DruckA_St_1       := L     21.3,
           i_CTRL_DruckA_St_2       := L     21.4,
           i_CTRL_DruckA_St_3       := L     21.5,
           i_CTRL_DruckA_St_4       := L     21.6,
           i_CTRL_DruckB_St_1       := L     21.7,
           i_CTRL_DruckB_St_2       := L     22.0,
           i_CTRL_DruckB_St_3       := L     22.1,
           i_CTRL_DruckB_St_4       := L     22.2,
           io_FM_Entspan_St_1_CTRL  := #dummy,
           io_FM_Entspan_St_2_CTRL  := #dummy,
           io_FM_Entspan_St_3_CTRL  := #dummy,
           io_FM_Entspan_St_4_CTRL  := #dummy,
           io_FM_Entspan_St_1_HAWE  := #dummy,
           io_FM_Entspan_St_2_HAWE  := #dummy,
           io_FM_Entspan_St_3_HAWE  := #dummy,
           io_FM_Entspan_St_4_HAWE  := #dummy);
      NOP   0;
NETWORK
TITLE =ProfiBus-AUSGANG-HAWE: DB_HR-Bereich an HAWE senden

      U     "m_null";
      =     L     21.0;
      BLD   103;
      U     "m_eins";
      =     L     21.1;
      BLD   103;
      CALL "FC_UT_IO_PROFIBUS" (
           read                     := L     21.0,
           write                    := L     21.1,
           Datenbereich             := "DB_HR".HAWE.an,
           Profibus_ADR             := "DB_CONFIG".ProfiBus.StartAdrPLC.OUT_HAWEBOX);
      NOP   0;
NETWORK
TITLE =M-Ausgang: SpannHydraulik Pumpe ein
